# B&R Automation Studio project Teknologia25 (part 8)

#### Main.cpp - Init, cyclic, exit code
```cpp
#include <bur/plctypes.h>
#ifdef _DEFAULT_INCLUDES
	#include <AsDefault.h>
#endif
#include <cosyWriteApi.h>
#include <cosyReadApi.h>
#include <stdint.h>
#include <stdio.h>
#include <parson.h>
#include <moApi.h>

#define TRUE 1
#define FALSE 0
#define booltoa(x) ((x)?"true":"false")

void cosyExample_ReadConfig(UDINT);
void cosyExample_WriteConfig(UDINT);
int json_get_array_memberStr(UDINT,UDINT,UDINT,int,UDINT);
int json_get_array_memberNumber(UDINT,UDINT,UDINT,int,UDINT);
int json_get_array_memberBool(UDINT,UDINT,UDINT,int,UDINT);
int json_dotget_number(UDINT,UDINT,UDINT);
unsigned long bur_heap_size = 0xffff;

void _INIT ProgramInit(void)
{
	webservice.enable = TRUE;
	webservice.pRequestHeader = (UDINT)&requestHeader;
	webservice.pRequestData = (UDINT)&request;
	webservice.requestDataSize = sizeof(request);
	webservice.pServiceName 	= (UDINT)&"conf6d.cgi"; //
	webservice.option 		= httpOPTION_HTTP_11 + httpOPTION_SERVICE_TYPE_NAME;

	webservice.pUri = (UDINT)&uri;
	webservice.uriSize = sizeof(uri);
	cosyExample_ReadConfig((UDINT)&layout);
}

void _CYCLIC ProgramCyclic(void)
{
	if(webservice.send)
	{
		webservice.send = FALSE;
	}
	else if(webservice.status == ERR_OK && webservice.phase == httpPHASE_RECEIVED && !webservice.send)
	{
		httpGetParamUrl_0.pSrc = (UDINT)&uri;
		httpGetParamUrl_0.enable = TRUE;
		httpGetParamUrl_0.pParam = (UDINT)&"cmd";
		httpGetParamUrl_0.pValue = (UDINT)&cmd;
		httpGetParamUrl_0.valueSize = sizeof(cmd);
		httpGetParamUrl(&httpGetParamUrl_0);

		if(httpGetParamUrl_0.status == ERR_OK)
		{
			httpGetParamUrl_0.enable = FALSE;
			httpGetParamUrl(&httpGetParamUrl_0);
		}

		if(brsstrcmp((UDINT)&cmd,(UDINT)&"read") == 0)
		{
			brsstrcpy((UDINT)&responseHeader.contentType,(UDINT)&"application/json");
			brsstrcpy((UDINT)&response,(UDINT)&"{\"status\":\"ok\",\"layout\":{\"x\":");
			sprintf(response,"%s%i,\"y\":%i,\"segments\":[",response,layout.Xcount,layout.Ycount);
			for(int i = 0; i < layout.SegmentCount; ++i)
			{
				sprintf(response,"%s{\"x\":%i,\"y\":%i,\"name\":\"%s\",\"IsMaster\":%s}",response,layout.Segments[i].x,layout.Segments[i].y,layout.Segments[i].Name,booltoa(layout.Segments[i].IsMaster));
				if(i != (layout.SegmentCount-1))
				{
					brsstrcat((UDINT)&response,(UDINT)&",");
				}
			}
			brsstrcat((UDINT)&response,(UDINT)&"]}}");
		}
		else if(brsstrcmp((UDINT)&cmd,(UDINT)&"write") == 0)
		{
			brsstrcpy((UDINT)&responseHeader.contentType,(UDINT)&"application/json");
			brsmemset((UDINT)&layout,0,sizeof(layout));
			json_dotget_number((UDINT)&request,(UDINT)&"x",(UDINT)&tmpREAL);
			layout.Xcount = (USINT)tmpREAL;
			json_dotget_number((UDINT)&request,(UDINT)&"y",(UDINT)&tmpREAL);
			layout.Ycount = (USINT)tmpREAL;
			layout.SegmentCount = 0;
			for(int i = 0; i < 255; ++i)
			{
				if(json_get_array_memberNumber((UDINT)&request,(UDINT)&"segments",(UDINT)&"x",i,(UDINT)&tmpREAL) >= 0)
				{
					layout.Segments[i].x = (INT)tmpREAL;
					json_get_array_memberNumber((UDINT)&request,(UDINT)&"segments",(UDINT)&"y",i,(UDINT)&tmpREAL);
					layout.Segments[i].y = (INT)tmpREAL;
					json_get_array_memberBool((UDINT)&request,(UDINT)&"segments",(UDINT)&"IsMaster",i,(UDINT)&layout.Segments[i].IsMaster);
					layout.SegmentCount++;
				}
				else
				{
					break;
				}
			}
			cosyExample_WriteConfig((UDINT)&layout);
			brsstrcpy((UDINT)&response,(UDINT)&"{\"status\":\"ok\"}");
		}
		else
		{
			brsstrcpy((UDINT)&responseHeader.contentType,(UDINT)&"image/svg+xml"); //
			httpDecodeBase64_0.enable = TRUE;
			httpDecodeBase64_0.destSize = sizeof(response);
			httpDecodeBase64_0.pDest = (UDINT)&response;
			httpDecodeBase64_0.pSrc = (UDINT)&svgResource;
			httpDecodeBase64_0.srcLen = brsstrlen((UDINT)&svgResource);
			httpDecodeBase64(&httpDecodeBase64_0);
		}
		brsstrcpy((UDINT)&responseHeader.userLine[0].name,(UDINT)&"Cross-Origin-Resource-Policy");
		brsstrcpy((UDINT)&responseHeader.userLine[0].value,(UDINT)&"cross-origin");
		brsstrcpy((UDINT)&responseHeader.userLine[1].name,(UDINT)&"Access-Control-Allow-Origin");
		brsstrcpy((UDINT)&responseHeader.userLine[1].value,(UDINT)&"*");
		webservice.pResponseHeader = (UDINT)&responseHeader;
		webservice.pResponseData = (UDINT)&response;
		webservice.responseDataLen 	= brsstrlen((UDINT)&response);
		webservice.send = TRUE;
	}
	httpService(&webservice);

}

/* In the example code, error handling was deliberately omitted. */
void cosyExample_ReadConfig(UDINT context)
{
	Layout_typ myLayout;
	brsmemcpy((UDINT)&myLayout,context,sizeof(myLayout));
	uint32_t intValue = 0;
	BOOL boolValue = FALSE;
	char strValue[130];
	char tempID[60];
	COSY_H hCosy = cosyOpenElement("System/mapp6D/LayoutConfiguration", "Layout6D_1");
	cosyGetPropertyValue(hCosy, "Segments/SegRow", "USINT", sizeof(intValue),&intValue, NULL);
	myLayout.Ycount = (USINT)intValue;
	cosyGetPropertyValue(hCosy, "Segments/SegCol", "USINT", sizeof(intValue),&intValue, NULL);
	myLayout.Xcount = (USINT)intValue;
	myLayout.SegmentCount = 0;
	for(int i = 0; i < 255; ++i)
	{
		sprintf(tempID,"Segments/Segment[%i]/X",(i+1));
		if(cosyGetPropertyValue(hCosy,tempID, "INT", sizeof(intValue),&intValue, NULL))
		{
			myLayout.Segments[i].x = (INT)intValue;
			sprintf(tempID,"Segments/Segment[%i]/Y",(i+1));
			cosyGetPropertyValue(hCosy,tempID, "INT", sizeof(intValue),&intValue, NULL);
			myLayout.Segments[i].y = (INT)intValue;
			sprintf(tempID,"Segments/Segment[%i]/Name",(i+1));
			cosyGetPropertyValue(hCosy,tempID, "STRING", sizeof(strValue),&strValue, NULL);
			brsstrcpy((UDINT)&myLayout.Segments[i].Name,(UDINT)&strValue);
			sprintf(tempID,"Segments/Segment[%i]/IsMaster",(i+1));
			cosyGetPropertyValue(hCosy,tempID, "BOOL", sizeof(intValue),&intValue, NULL);
			myLayout.Segments[i].IsMaster = (BOOL)intValue;
			myLayout.SegmentCount++;
		}
		else
		{
			break;
		}
	}
	cosyCloseElement(hCosy);
	brsmemcpy(context,(UDINT)&myLayout,sizeof(myLayout));
}
void cosyExample_WriteConfig(UDINT context)
{
	Layout_typ myLayout;
	uint32_t intValue = 0;
	BOOL boolValue = FALSE;
	USINT usintValue = 0;
	USINT i = 0;
	INT tempINT = 0;
	DINT tempDINT = 0;
	char segmentName[60];
	brsmemcpy((UDINT)&myLayout,context,sizeof(myLayout));
	COSY_H hCosy = cosyOpenElement("System/mapp6D/LayoutConfiguration", "Layout6D_1");
	if(hCosy != NULL)
	{
		cosySetProperty(hCosy, "Segments/SegCol", "USINT", &myLayout.Xcount, sizeof(myLayout.Xcount));
		cosySetProperty(hCosy, "Segments/SegRow", "USINT", &myLayout.Ycount, sizeof(myLayout.Ycount));
		for(i = 0; i < 255; ++i)
		{
			sprintf(segmentName,"Segments/Segment[%i]",(i+1));
			if(!cosyDeleteMember(hCosy,segmentName,COSY_TIMEOUT_NO_WAIT))
			{
				break;
			}
		}
		for(i = 0; i < myLayout.SegmentCount; ++i)
		{
			sprintf(segmentName,"Segments/Segment[%i]",(i+1));
			cosyAddGroup(hCosy, segmentName, NULL);

			sprintf(segmentName,"Segments/Segment[%i]/Y",(i+1));
			cosySetProperty(hCosy, segmentName, "INT", &myLayout.Segments[i].y, sizeof(myLayout.Segments[i].y));
			sprintf(segmentName,"Segments/Segment[%i]/X",(i+1));
			cosySetProperty(hCosy, segmentName, "INT", &myLayout.Segments[i].x, sizeof(myLayout.Segments[i].x));
			sprintf(segmentName,"Segments/Segment[%i]/Name",(i+1));
			cosySetProperty(hCosy, segmentName, "STRING", &myLayout.Segments[i].Name, sizeof(myLayout.Segments[i].Name));
			sprintf(segmentName,"Segments/Segment[%i]/IsMaster",(i+1));

			cosySetProperty(hCosy, segmentName, "BOOL", &myLayout.Segments[i].IsMaster, 0);

			sprintf(segmentName,"Segments/Segment[%i]/PowerSectorName",(i+1));
			cosySetProperty(hCosy, segmentName, "STRING", "", 0);
			sprintf(segmentName,"Segments/Segment[%i]/Gaps",(i+1));
			cosyAddGroup(hCosy, segmentName, NULL);
			tempDINT = 0;
			sprintf(segmentName,"Segments/Segment[%i]/Gaps/Left",(i+1));
			cosySetProperty(hCosy, segmentName, "DINT", &tempDINT,sizeof(tempDINT));
			sprintf(segmentName,"Segments/Segment[%i]/Gaps/Bottom",(i+1));
			cosySetProperty(hCosy, segmentName, "DINT", &tempDINT,sizeof(tempDINT));
			sprintf(segmentName,"Segments/Segment[%i]/Gaps/Right",(i+1));
			cosySetProperty(hCosy, segmentName, "DINT", &tempDINT,sizeof(tempDINT));
			sprintf(segmentName,"Segments/Segment[%i]/Gaps/Top",(i+1));
			cosySetProperty(hCosy, segmentName, "DINT", &tempDINT,sizeof(tempDINT));
		}
		cosySaveElement(hCosy);
		cosyCloseElement(hCosy);
	}
}

int json_get_array_memberStr(UDINT data,UDINT arraystr,UDINT target,int index,UDINT result)
{
	/*TODO: Add your code here*/
	char buf[8000];
	char member[32];
	char memberValue[256];
	brsstrcpy((UDINT)&buf,data);

	JSON_Value *jsonRoot = json_parse_string(buf);
	brsstrcpy((UDINT)&member,arraystr);
	int retVal = 0;
	if(jsonRoot != NULL)
	{
		JSON_Array *arr = json_object_dotget_array(json_object(jsonRoot), member);
		if(arr != NULL)
		{
			JSON_Object *arrValue = json_array_get_object(arr,(size_t)index);
			if(arrValue != NULL)
			{
				const char *tempStr = NULL;
				char test[30];
				brsstrcpy((UDINT)&test,target);
				tempStr = json_object_dotget_string(arrValue,test);
				if(tempStr != NULL)
				{
					brsstrcpy(result,(UDINT)tempStr);
					retVal = 0;
				}
				else
				{
					retVal = -1;
				}
			}
			else
			{
				retVal = -1;
			}
		}
		else
		{
			retVal = -1;
		}
	}
	else
	{
		retVal = -1;
	}

	json_value_free(jsonRoot);
	return retVal;
}

int json_get_array_memberNumber(UDINT data,UDINT arraystr,UDINT target,int index,UDINT result)
{
	/*TODO: Add your code here*/
	char buf[8000];
	char member[32];
	char memberValue[256];
	brsstrcpy((UDINT)&buf,data);

	JSON_Value *jsonRoot = json_parse_string(buf);
	brsstrcpy((UDINT)&member,arraystr);
	int retVal = 0;
	if(jsonRoot != NULL)
	{
		JSON_Array *arr = json_object_dotget_array(json_object(jsonRoot), member);
		if(arr != NULL)
		{
			JSON_Object *arrValue = json_array_get_object(arr,(size_t)index);
			if(arrValue != NULL)
			{
				char test[30];
				brsstrcpy((UDINT)&test,target);
				double number = json_object_dotget_number(arrValue,test);
				REAL tempREAL = (REAL)number;
				brsmemcpy(result,(UDINT)&tempREAL,sizeof(tempREAL));
				//brsstrcpy(result,(UDINT)tempStr);
				retVal = 0;
			}
			else
			{
				retVal = -1;
			}
		}
		else
		{
			retVal = -1;
		}
	}
	else
	{
		retVal = -1;
	}

	json_value_free(jsonRoot);
	return retVal;
}

int json_get_array_memberBool(UDINT data,UDINT arraystr,UDINT target,int index,UDINT result)
{
	/*TODO: Add your code here*/
	char buf[8000];
	char member[32];
	char memberValue[256];
	brsstrcpy((UDINT)&buf,data);

	JSON_Value *jsonRoot = json_parse_string(buf);
	brsstrcpy((UDINT)&member,arraystr);
	int retVal = 0;
	if(jsonRoot != NULL)
	{
		JSON_Array *arr = json_object_dotget_array(json_object(jsonRoot), member);
		if(arr != NULL)
		{
			JSON_Object *arrValue = json_array_get_object(arr,(size_t)index);
			if(arrValue != NULL)
			{
				char test[30];
				brsstrcpy((UDINT)&test,target);
				int number = json_object_dotget_boolean(arrValue,test);
				BOOL tempBOOL = (BOOL)number;
				brsmemcpy(result,(UDINT)&tempBOOL,sizeof(tempBOOL));
				//brsstrcpy(result,(UDINT)tempStr);
				retVal = 0;
			}
			else
			{
				retVal = -1;
			}
		}
		else
		{
			retVal = -1;
		}
	}
	else
	{
		retVal = -1;
	}
	json_value_free(jsonRoot);
	return retVal;
}

int json_dotget_number(UDINT data,UDINT memberstr,UDINT result)
{
	/*TODO: Add your code here*/
	char buf[8000];
	char member[32];
	char memberValue[256];
	brsstrcpy((UDINT)&buf,data);

	JSON_Value *jsonRoot = json_parse_string(buf);
	brsstrcpy((UDINT)&member,memberstr);
	int retVal = -1;
	if(jsonRoot != NULL)
	{
		double temp = 0;
		temp = json_object_dotget_number(json_object(jsonRoot), member);
		REAL tempREAL = (REAL)temp;
		brsmemcpy(result,(UDINT)&tempREAL,sizeof(tempREAL));
		retVal = 0;
		//memcpy(result,(UDINT)&temp,4);

	}

	json_value_free(jsonRoot);
	return retVal;
}
```

#### Types.typ - Local data types
```iecst
TYPE
	Segment_typ : 	STRUCT
		x : INT;
		y : INT;
		IsMaster : BOOL;
		Name : STRING[20];
	END_STRUCT;
	Layout_typ : 	STRUCT
		Segments : ARRAY[0..99]OF Segment_typ;
		SegmentCount : USINT;
		Xcount : USINT;
		Ycount : USINT;
	END_STRUCT;
END_TYPE
```

#### Variables.var - Local variables
```iecst
VAR
	layout : Layout_typ;
	webservice : httpService;
	httpDecodeBase64_0 : httpDecodeBase64;
	requestHeader : httpRequestHeader_t;
	responseHeader : httpResponseHeader_t;
	svgResource : STRING[13500] := 'PHN2ZyBpZD0iNmRzdmciIHhtbG5zPSJodHRwOi8vd3d3LnczLm9yZy8yMDAwL3N2ZyIgd2lkdGg9IjYwMCIgaGVpZ2h0PSI4MjAiIHhtbDpzcGFjZT0icHJlc2VydmUiIGNvbG9yLWludGVycG9sYXRpb24tZmlsdGVycz0ic1JHQiI+Cgk8c3R5bGU+c3Zne2ZpbGw6bm9uZTsgZmlsbCAtIHJ1bGU6ZXZlbm9kZDsgZm9udCAtIHNpemU6MTJweDsgb3ZlcmZsb3c6dmlzaWJsZTsgc3Ryb2tlIC0gbGluZWNhcDpzcXVhcmU7IHN0cm9rZSAtIG1pdGVybGltaXQ6Mzt9LnNlZ21lbnQucG93ZXItb2ZmIHtmaWxsOnJnYigyNTMsIDI1MywgMjUzKTt9LnNlZ21lbnQucG93ZXItb24ge2ZpbGw6cmdiKDE0NiwgMjA4LCA4MCk7fS5zZWdtZW50LmVycm9yIHtmaWxsOnJnYigyNTIsIDIyLCAxNik7fS5zZWdtZW50ICZndDsgcmVjdCB7c3Ryb2tlOiM1OTU5NTk7c3Ryb2tlLWxpbmVjYXA6cm91bmQ7c3Ryb2tlLWxpbmVqb2luOnJvdW5kO3N0cm9rZS13aWR0aDozLjc1MDAwMDt9IC5zaHV0dGxlICZndDsgZyAmZ3Q7IHJlY3Qge3N0cm9rZTpibGFjaztzdHJva2UtbGluZWNhcDpyb3VuZDtzdHJva2UtbGluZWpvaW46cm91bmQ7c3Ryb2tlLXdpZHRoOjUuMDAwMDtmaWxsOmxpZ2h0Z3JheTt9IC5zaHV0dGxlLndhcm5pbmcgJmd0OyBnICZndDsgcmVjdCB7ZmlsbDp5ZWxsb3c7fSAuc2h1dHRsZS5lcnJvciAmZ3Q7IGcgJmd0OyByZWN0IHtmaWxsOnJlZDt9IC5zaHV0dGxlLmRpc2FibGVkICZndDsgZyAmZ3Q7IHJlY3Qge2ZpbGw6Z3JheTt9IC5zaHV0dGxlLmRpc2NvdmVyaW5nICZndDsgZyAmZ3Q7IHJlY3Qge2ZpbGw6ZGFya29yYW5nZTt9ICAuc21hbGwge2ZvbnQ6IDE1cHggc2Fucy1zZXJpZjtjb2xvcjpibGFjaztzdHJva2U6YmxhY2s7ZmlsbDpibGFjazstd2Via2l0LXVzZXItc2VsZWN0OiBub25lOyAtbXMtdXNlci1zZWxlY3Q6IG5vbmU7IHVzZXItc2VsZWN0OiBub25lO30gLnNodXR0bGV7IGN1cnNvcjpwb2ludGVyfSAuc2h1dHRsZTphY3RpdmUgJmd0OyBnICZndDsgcmVjdCB7ZmlsbDpsaWdodGJsdWU7fSAuc2h1dHRsZS50ZW1wICZndDsgZyAmZ3Q7IHJlY3Qge2ZpbGw6cmdiYSgxMjcsMTI3LDEyNywwLjEpO3N0cm9rZTpyZ2JhKDAsMCwwLDAuMSk7c3Ryb2tlLWRhc2hhcnJheToyMDt9IC5zaHV0dGxlLnRlbXAuYWN0aXZlICZndDsgZyAmZ3Q7IHJlY3Qge2ZpbGw6cmdiYSgxMjcsMCwwLDAuMSk7fTwvc3R5bGU+Cgk8cmVjdCB4PSI0OCIgeT0iMjMiIHN0eWxlPSJzdHJva2U6bGlnaHRncmF5O3N0cm9rZS13aWR0aDoxcHgiIHdpZHRoPSI0ODQiIGhlaWdodD0iMTA1Ii8+Cgk8Zm9yZWlnbk9iamVjdCB4PSIxMDAiIHk9IjM1IiAKCQkJCXdpZHRoPSI1MDAiIGhlaWdodD0iMTYwIiA+IAoJCTxkaXYgeG1sbnM9Imh0dHA6Ly93d3cudzMub3JnLzE5OTkveGh0bWwiPiAKCQkJPGxhYmVsIGZvcj0ieFNpemUiPlggRGlyZWN0aW9uPC9sYWJlbD48YnIvPgoJCQk8aW5wdXQgdHlwZT0ibnVtYmVyIiBpZD0ieFNpemUiIG5hbWU9InhTaXplIiBtaW49IjEiIG1heD0iMzAiIHZhbHVlPSIxIiAvPgkJCQoJCTwvZGl2PiAKCTwvZm9yZWlnbk9iamVjdD4gCgk8Zm9yZWlnbk9iamVjdCB4PSIyNTAiIHk9IjM1IiAKCQkJCXdpZHRoPSI1MDAiIGhlaWdodD0iMTYwIiA+IAoJCTxkaXYgeG1sbnM9Imh0dHA6Ly93d3cudzMub3JnLzE5OTkveGh0bWwiPiAKCQkJPGxhYmVsIGZvcj0ieVNpemUiPlkgRGlyZWN0aW9uPC9sYWJlbD48YnIvPgoJCQk8aW5wdXQgdHlwZT0ibnVtYmVyIiBpZD0ieVNpemUiIG5hbWU9InlTaXplIiBtaW49IjEiIG1heD0iMzAiIHZhbHVlPSIxIi8+CgkJPC9kaXY+IAoJPC9mb3JlaWduT2JqZWN0PiAKCTxmb3JlaWduT2JqZWN0IHg9IjM3NSIgeT0iMzUiIAoJCQkJd2lkdGg9IjExMCIgaGVpZ2h0PSIxNjAiID4gCgkJPGRpdiB4bWxucz0iaHR0cDovL3d3dy53My5vcmcvMTk5OS94aHRtbCI+IAoJCQk8bGFiZWwgPkFjdGl2ZSBTZWdtZW50czwvbGFiZWw+PGJyLz4KCQkJPGNlbnRlcj48bGFiZWwgaWQ9InNlZ21lbnRDb3VudCI+MDwvbGFiZWw+PC9jZW50ZXI+CgkJPC9kaXY+IAoJPC9mb3JlaWduT2JqZWN0PiAKCTxmb3JlaWduT2JqZWN0IHg9IjM2NSIgeT0iOTUiIAoJCQkJd2lkdGg9IjI1MCIgaGVpZ2h0PSIxNjAiID4gCgkJPGRpdiB4bWxucz0iaHR0cDovL3d3dy53My5vcmcvMTk5OS94aHRtbCI+IAoJCQk8YnV0dG9uIHR5cGU9ImJ1dHRvbiIgb25jbGljaz0icmVhZFBMQygpIj5SZWFkIFBMQzwvYnV0dG9uPgoJCQk8YnV0dG9uIHR5cGU9ImJ1dHRvbiIgb25jbGljaz0id3JpdGVQTEMoKSI+V3JpdGUgUExDPC9idXR0b24+CgkJPC9kaXY+IAoJPC9mb3JlaWduT2JqZWN0PiAKCTxnIGlkPSJnQXNzZW1ibHk2RF8xIiBjbGFzcz0iYXNzZW1ibHkiIHRyYW5zZm9ybT0idHJhbnNsYXRlKDUwLjAwMDAwMCA2MjAuMDAwMDAwKSI+CgkJPGcgaWQ9IkxheW91dDZEXzEiIGNsYXNzPSJsYXlvdXQiPgoJCQk8ZyBpZD0ic2VnbWVudHMiPjwvZz4KCQk8L2c+Cgk8L2c+Cgk8ZyBpZD0iY29udGV4dE1lbnUiPjwvZz4KCTxzY3JpcHQ+Ly88IVtDREFUQVsKCQl2YXIgeENvdW50ID0gZG9jdW1lbnQuZ2V0RWxlbWVudEJ5SWQoJ3hTaXplJyk7CgkJdmFyIHlDb3VudCA9IGRvY3VtZW50LmdldEVsZW1lbnRCeUlkKCd5U2l6ZScpOwoJCXZhciBzZWdtZW50cyA9IGRvY3VtZW50LmdldEVsZW1lbnRCeUlkKCdzZWdtZW50cycpOwoJCXZhciBzZWdtZW50Q291bnQgPSBkb2N1bWVudC5nZXRFbGVtZW50QnlJZCgnc2VnbWVudENvdW50Jyk7CgkJdmFyIGNvbnRleHRNZW51ID0gZG9jdW1lbnQuZ2V0RWxlbWVudEJ5SWQoJ2NvbnRleHRNZW51Jyk7CgkJdmFyIHNlZ21lbnRTaXplID0gMDsKCQl4Q291bnQuYWRkRXZlbnRMaXN0ZW5lcigiY2hhbmdlIiwgKGV2ZW50KSA9PiB7c2V0TGF5b3V0KHhDb3VudC52YWx1ZSx5Q291bnQudmFsdWUpO30pOwoJCXlDb3VudC5hZGRFdmVudExpc3RlbmVyKCJjaGFuZ2UiLCAoZXZlbnQpID0+IHtzZXRMYXlvdXQoeENvdW50LnZhbHVlLHlDb3VudC52YWx1ZSk7fSk7CgkJCgkJdmFyIGFjdGl2ZVNlZ21lbnRzID0gW107CgkJdmFyIHN2Z0VsZW0gPSBkb2N1bWVudC5nZXRFbGVtZW50QnlJZCgnNmRzdmcnKTsKCQkJCXN2Z0VsZW0uYWRkRXZlbnRMaXN0ZW5lcigibG9hZCIsICgpID0+IHsKCQkJcmVhZFBMQygpOwoJCX0pOwoJCWZ1bmN0aW9uIHJlYWRQTEMoKQoJCXsKCQkJdmFyIHhodHRwID0gbmV3IFhNTEh0dHBSZXF1ZXN0KCk7CgkJCQl4aHR0cC5vbnJlYWR5c3RhdGVjaGFuZ2UgPSBmdW5jdGlvbigpIHsKCQkJCQlpZiAodGhpcy5yZWFkeVN0YXRlID09IDQgJiYgdGhpcy5zdGF0dXMgPT0gMjAwKSB7CgkJCQkJICAgLy8gVHlwaWNhbCBhY3Rpb24gdG8gYmUgcGVyZm9ybWVkIHdoZW4gdGhlIGRvY3VtZW50IGlzIHJlYWR5OgoJCQkJCSAgIHZhciBkYXRhID0gSlNPTi5wYXJzZSh4aHR0cC5yZXNwb25zZVRleHQpOwoJCQkJCSAgIGFjdGl2ZVNlZ21lbnRzID0gW107CgkJCQkJICAgZm9yKHZhciBpID0gMDsgaSA8IGRhdGEubGF5b3V0LnNlZ21lbnRzLmxlbmd0aDsgKytpKQoJCQkJCSAgIHsKCQkJCQkJCWFjdGl2ZVNlZ21lbnRzLnB1c2goe3g6ZGF0YS5sYXlvdXQuc2VnbWVudHNbaV0ueCx5OmRhdGEubGF5b3V0LnNlZ21lbnRzW2ldLnksSXNNYXN0ZXI6ZGF0YS5sYXlvdXQuc2VnbWVudHNbaV0uSXNNYXN0ZXJ9KTsKCQkJCQkJCWlmKGRhdGEubGF5b3V0LnNlZ21lbnRzW2ldLklzTWFzdGVyKQoJCQkJCQkJewoJCQkJCQkJCXNldE1hc3RlckJ5U2VnbWVudChhY3RpdmVTZWdtZW50c1thY3RpdmVTZWdtZW50cy5sZW5ndGgtMV0pOwoJCQkJCQkJfQoJCQkJCSAgIH0KCQkJCQkgICB4Q291bnQudmFsdWUgPSBkYXRhLmxheW91dC54OwoJCQkJCSAgIHlDb3VudC52YWx1ZSA9IGRhdGEubGF5b3V0Lnk7CgkJCQkJICAgc2V0TGF5b3V0KGRhdGEubGF5b3V0LngsZGF0YS5sYXlvdXQueSk7CgkJCQkJfQoJCQkJfTsKCQkJCXhodHRwLm9wZW4oIkdFVCIsICIvY29uZjZkLmNnaT9jbWQ9cmVhZCIsIHRydWUpOwoJCQkJeGh0dHAuc2VuZCgpOwoJCX0KCQlmdW5jdGlvbiB3cml0ZVBMQygpCgkJewoJCQl2YXIgeGh0dHAgPSBuZXcgWE1MSHR0cFJlcXVlc3QoKTsKCQkJCXhodHRwLm9ucmVhZHlzdGF0ZWNoYW5nZSA9IGZ1bmN0aW9uKCkgewoJCQkJCWlmICh0aGlzLnJlYWR5U3RhdGUgPT0gNCAmJiB0aGlzLnN0YXR1cyA9PSAyMDApIHsKCQkJCQkgICAvLyBUeXBpY2FsIGFjdGlvbiB0byBiZSBwZXJmb3JtZWQgd2hlbiB0aGUgZG9jdW1lbnQgaXMgcmVhZHk6CgkJCQkJICAgdmFyIGRhdGEgPSBKU09OLnBhcnNlKHhodHRwLnJlc3BvbnNlVGV4dCk7CgkJCQkJICAgY29uc29sZS5sb2coZGF0YSk7CgkJCQkJfQoJCQkJfTsKCQkJCXhodHRwLm9wZW4oIlBPU1QiLCAiL2NvbmY2ZC5jZ2k/Y21kPXdyaXRlIiwgdHJ1ZSk7CgkJCQlhY3RpdmVTZWdtZW50cy5zb3J0KGNvbXBhcmVGbik7CgkJCQl2YXIgbWFzdGVyRWxlbWVudCA9IGRvY3VtZW50LmdldEVsZW1lbnRCeUlkKCdtYXN0ZXItdGV4dCcpOwoJCQkJaWYoIW1hc3RlckVsZW1lbnQpCgkJCQl7CgkJCQkJYWN0aXZlU2VnbWVudHNbMF0uSXNNYXN0ZXIgPSB0cnVlOwoJCQkJfQoJCQkJeGh0dHAuc2VuZChKU09OLnN0cmluZ2lmeSh7eDpwYXJzZUludCh4Q291bnQudmFsdWUpLHk6cGFyc2VJbnQoeUNvdW50LnZhbHVlKSxzZWdtZW50czphY3RpdmVTZWdtZW50c30pKTsKCQl9CgkJCgkJZnVuY3Rpb24gY29tcGFyZUZuKGEsIGIpIHsKCQkgIGlmIChhLnggPCBiLngpIHsKCQkJcmV0dXJuIC0xOwoJCSAgfWVsc2UgaWYgKGEueCA+IGIueCkgewoJCQlyZXR1cm4gMTsKCQkgIH1lbHNlIGlmIChhLnkgPCBiLnkpIHsKCQkJcmV0dXJuIC0xOwoJCSAgfWVsc2UgaWYgKGEueSA+IGIueSkgewoJCQlyZXR1cm4gMTsKCQkgIH0KCQkgIC8vIGEgbXVzdCBiZSBlcXVhbCB0byBiCgkJICByZXR1cm4gMDsKCQl9OwoJCQoJCWZ1bmN0aW9uIGNoYW5nZVN0eWxlKHRoYXQpCgkJewoJCQlpZihjb250ZXh0TWVudS5pbm5lckhUTUwgPT0gJycpCgkJCXsKCQkJCWlmKHRoYXQuY2xhc3NMaXN0WzFdID09ICdwb3dlci1vZmYnKQoJCQkJewoJCQkJCXRoYXQuY2xhc3NMaXN0LnJlbW92ZSgicG93ZXItb2ZmIik7CgkJCQkJdGhhdC5jbGFzc0xpc3QuYWRkKCJwb3dlci1vbiIpOwoJCQkJCWFjdGl2ZVNlZ21lbnRzLnB1c2goe3g6cGFyc2VJbnQodGhhdC5nZXRBdHRyaWJ1dGUoJ3Bvc2l0aW9uLXgnKSkseTpwYXJzZUludCh0aGF0LmdldEF0dHJpYnV0ZSgncG9zaXRpb24teScpKSxJc01hc3RlcjpmYWxzZX0pOwoJCQkJfQoJCQkJZWxzZQoJCQkJewoJCQkJCXRoYXQuY2xhc3NMaXN0LmFkZCgicG93ZXItb2ZmIik7CgkJCQkJdGhhdC5jbGFzc0xpc3QucmVtb3ZlKCJwb3dlci1vbiIpOwoJCQkJCXZhciByZW1vdmVJdGVtID0ge3g6dGhhdC5nZXRBdHRyaWJ1dGUoJ3Bvc2l0aW9uLXgnKSx5OnRoYXQuZ2V0QXR0cmlidXRlKCdwb3NpdGlvbi15Jyl9CgkJCQkJZm9yKHZhciBpID0gMDsgaSA8IGFjdGl2ZVNlZ21lbnRzLmxlbmd0aDsgKytpKQoJCQkJCXsKCQkJCQkJaWYoKGFjdGl2ZVNlZ21lbnRzW2ldLnggPT0gcmVtb3ZlSXRlbS54KSAmJiAoYWN0aXZlU2VnbWVudHNbaV0ueSA9PSByZW1vdmVJdGVtLnkpKQoJCQkJCQl7CgkJCQkJCQlhY3RpdmVTZWdtZW50cy5zcGxpY2UoaSwgMSk7CgkJCQkJCQlicmVhazsKCQkJCQkJfQoJCQkJCX0KCQkJCX0KCQkJfQoJCQljb250ZXh0TWVudS5pbm5lckhUTUwgPSAnJzsKCQkJc2VnbWVudENvdW50LmlubmVySFRNTCA9IGFjdGl2ZVNlZ21lbnRzLmxlbmd0aDsKCQkJCgkJfQoJCWZ1bmN0aW9uIHNldE1hc3Rlcih0aGF0KQoJCXsKCQkJdmFyIGlkeCA9IHBhcnNlSW50KHRoYXQuZ2V0QXR0cmlidXRlKCdzZWdtZW50LWluZGV4JykpOwoJCQl2YXIgdGFyZ2V0SWQgPSB0aGF0LmdldEF0dHJpYnV0ZSgndGFyZ2V0LWlkJyk7CgkJCWZvcih2YXIgaSA9IDA7IGkgPCBhY3RpdmVTZWdtZW50cy5sZW5ndGg7ICsraSkKCQkJewoJCQkJYWN0aXZlU2VnbWVudHNbaV1bIklzTWFzdGVyIl0gPSBmYWxzZTsKCQkJfQoJCQlhY3RpdmVTZWdtZW50c1tpZHhdWyJJc01hc3RlciJdID0gdHJ1ZTsKCQkJY29udGV4dE1lbnUuaW5uZXJIVE1MID0gJyc7CgkJCQoJCQl2YXIgdGFyZ2V0ID0gZG9jdW1lbnQuZ2V0RWxlbWVudEJ5SWQodGFyZ2V0SWQpOwoJCQl2YXIgbWFzdGVyVGV4dCA9IGRvY3VtZW50LmdldEVsZW1lbnRCeUlkKCdtYXN0ZXItdGV4dCcpOwoJCQlpZihtYXN0ZXJUZXh0KQoJCQl7CgkJCQltYXN0ZXJUZXh0LnBhcmVudEVsZW1lbnQucmVtb3ZlQ2hpbGQobWFzdGVyVGV4dCk7CgkJCX0KCQkJdmFyIHRleHQgPSBkb2N1bWVudC5jcmVhdGVFbGVtZW50TlMoImh0dHA6Ly93d3cudzMub3JnLzIwMDAvc3ZnIiwgInRleHQiKTsKCQkJdGV4dC5zZXRBdHRyaWJ1dGUoJ3gnLDUpOwoJCQl0ZXh0LnNldEF0dHJpYnV0ZSgneScsMTgpOwoJCQl0ZXh0LnNldEF0dHJpYnV0ZSgnc3R5bGUnLCdmaWxsOndoaXRlO2ZvbnQtc2l6ZToxOHB4OycpOwoJCQl0ZXh0LnNldEF0dHJpYnV0ZSgnaWQnLCdtYXN0ZXItdGV4dCcpOwoJCQl0ZXh0LmlubmVySFRNTCA9ICdNJzsKCQkJdGFyZ2V0LmFwcGVuZENoaWxkKHRleHQpOwoJCX0KCQkKCQlmdW5jdGlvbiBzZXRNYXN0ZXJCeVNlZ21lbnQoc2VnbWVudCkKCQl7CgkJCXZhciBzZWxlY3RlZFNlZ21lbnRzID0gZG9jdW1lbnQuZ2V0RWxlbWVudHNCeUNsYXNzTmFtZSgnc2VnbWVudCBwb3dlci1vbicpOwoJCQlmb3IodmFyIGkgPSAwOyBpIDwgc2VsZWN0ZWRTZWdtZW50cy5sZW5ndGg7ICsraSkKCQkJewoJCQkJaWYoKHBhcnNlSW50KHNlbGVjdGVkU2VnbWVudHNbaV0uZ2V0QXR0cmlidXRlKCdwb3NpdGlvbi14JykpID09IHNlZ21lbnQueCkgJiYgKHBhcnNlSW50KHNlbGVjdGVkU2VnbWVudHNbaV0uZ2V0QXR0cmlidXRlKCdwb3NpdGlvbi15JykpID09IHNlZ21lbnQueSkpCgkJCQl7CgkJCQkJdmFyIG1hc3RlclRleHQgPSBkb2N1bWVudC5nZXRFbGVtZW50QnlJZCgnbWFzdGVyLXRleHQnKTsKCQkJCQlpZihtYXN0ZXJUZXh0KQoJCQkJCXsKCQkJCQkJbWFzdGVyVGV4dC5wYXJlbnRFbGVtZW50LnJlbW92ZUNoaWxkKG1hc3RlclRleHQpOwoJCQkJCX0KCQkJCQl2YXIgdGV4dCA9IGRvY3VtZW50LmNyZWF0ZUVsZW1lbnROUygiaHR0cDovL3d3dy53My5vcmcvMjAwMC9zdmciLCAidGV4dCIpOwoJCQkJCXRleHQuc2V0QXR0cmlidXRlKCd4Jyw1KTsKCQkJCQl0ZXh0LnNldEF0dHJpYnV0ZSgneScsMTgpOwoJCQkJCXRleHQuc2V0QXR0cmlidXRlKCdzdHlsZScsJ2ZpbGw6d2hpdGU7Zm9udC1zaXplOjE4cHg7Jyk7CgkJCQkJdGV4dC5zZXRBdHRyaWJ1dGUoJ2lkJywnbWFzdGVyLXRleHQnKTsKCQkJCQl0ZXh0LmlubmVySFRNTCA9ICdNJzsKCQkJCQlzZWxlY3RlZFNlZ21lbnRzW2ldLmFwcGVuZENoaWxkKHRleHQpOwoJCQkJCWJyZWFrOwoJCQkJfQoJCQl9CgkJfQoJCQoJCWZ1bmN0aW9uIGFkZENvbnRleHRtZW51KGV2ZW50KQoJCXsKCQkJdmFyIHNlZ21lbnRBY3RpdmUgPSBmYWxzZTsKCQkJdmFyIHNlZ21lbnRJbmRleCA9IDA7CgkJCWZvcih2YXIgaSA9IDA7IGkgPCBhY3RpdmVTZWdtZW50cy5sZW5ndGg7ICsraSkKCQkJewoJCQkJaWYoZXZlbnQudGFyZ2V0LnBhcmVudEVsZW1lbnQuZ2V0QXR0cmlidXRlKCdwb3NpdGlvbi14JykgPT0gYWN0aXZlU2VnbWVudHNbaV0ueCAmJiBldmVudC50YXJnZXQucGFyZW50RWxlbWVudC5nZXRBdHRyaWJ1dGUoJ3Bvc2l0aW9uLXknKSA9PSBhY3RpdmVTZWdtZW50c1tpXS55KQoJCQkJewoJCQkJCXNlZ21lbnRBY3RpdmUgPSB0cnVlOwoJCQkJCXNlZ21lbnRJbmRleCA9IGk7CgkJCQkJc2VnbWVudElkID0gZXZlbnQudGFyZ2V0LnBhcmVudEVsZW1lbnQuZ2V0QXR0cmlidXRlKCdpZCcpOwoJCQkJCWJyZWFrOwoJCQkJfQoJCQl9CgkJCWlmKGV2ZW50LnByZXZlbnREZWZhdWx0ICE9IHVuZGVmaW5lZCkKCQkJICBldmVudC5wcmV2ZW50RGVmYXVsdCgpOwoJCQkgaWYoZXZlbnQuc3RvcFByb3BhZ2F0aW9uICE9IHVuZGVmaW5lZCkKCQkJICBldmVudC5zdG9wUHJvcGFnYXRpb24oKTsKCQkJIGlmKHNlZ21lbnRBY3RpdmUpCgkJCSB7CgkJCQl2YXIgY21ZID0gZXZlbnQueS0xMDUvMjsKCQkJCWNvbnRleHRNZW51LmlubmVySFRNTCA9IGA8cmVjdCB4PSIke2V2ZW50Lnh9IiB5PSIke2NtWX0iIHN0eWxlPSJzdHJva2U6bGlnaHRncmF5O3N0cm9rZS13aWR0aDoxcHg7ZmlsbDp3aGl0ZTsiIHdpZHRoPSIxMDAiIGhlaWdodD0iMTA1Ii8+CgkJCSA8Zm9yZWlnbk9iamVjdCB4PSIke2V2ZW50LngrMn0iIHk9IiR7Y21ZfSIgCgkJCQkJCXdpZHRoPSI5NiIgaGVpZ2h0PSIxMDEiID4gCgkJCQkJCTxkaXYgeG1sbnM9Imh0dHA6Ly93d3cudzMub3JnLzE5OTkveGh0bWwiPiAKCQkJCQkJCTxidXR0b24gdHlwZT0iYnV0dG9uIiBvbmNsaWNrPSJzZXRNYXN0ZXIodGhpcykiIHNlZ21lbnQtaW5kZXg9IiR7c2VnbWVudEluZGV4fSIgdGFyZ2V0LWlkPSIke3NlZ21lbnRJZH0iPlNldCBhcyBNYXN0ZXI8L2J1dHRvbj4KCQkJCQkJPC9kaXY+IAoJCQkgPC9mb3JlaWduT2JqZWN0PiBgOwoJCQkgfQoJCX0KCQlmdW5jdGlvbiBzZXRMYXlvdXQoeCx5KQoJCXsKCQkJc2VnbWVudHMuaW5uZXJIVE1MID0gJyc7CgkJCXNlZ21lbnRTaXplID0gNDgwL3k7CgkJCWlmKHBhcnNlSW50KHgpID4gcGFyc2VJbnQoeSkpCgkJCXsKCQkJCXNlZ21lbnRTaXplID0gNDgwL3g7CgkJCX0KCQkJdmFyIHNlZ21lbnRDb3VudGVyID0gMTsKCQkJdmFyIGR5bkhXID0gJyc7CgkJCWZvcih2YXIgaSA9IDA7IGkgPCBhY3RpdmVTZWdtZW50cy5sZW5ndGg7ICsraSkKCQkJewoJCQkJaWYoKHBhcnNlSW50KGFjdGl2ZVNlZ21lbnRzW2ldLngpKzEpID4gcGFyc2VJbnQoeCkpCgkJCQl7CgkJCQkJYWN0aXZlU2VnbWVudHMuc3BsaWNlKGksMSk7CgkJCQkJaSA9IDA7CgkJCQkJY29udGludWU7CgkJCQl9CgkJCQlpZigocGFyc2VJbnQoYWN0aXZlU2VnbWVudHNbaV0ueSkrMSkgPiBwYXJzZUludCh5KSkKCQkJCXsKCQkJCQlhY3RpdmVTZWdtZW50cy5zcGxpY2UoaSwxKTsKCQkJCQlpID0gMDsKCQkJCQljb250aW51ZTsKCQkJCX0KCQkJfQoJCQlmb3IodmFyIGkgPSAwOyBpIDwgeDsgKytpKQoJCQl7CgkJCQlmb3IodmFyIGogPSAwOyBqIDwgeTsgKytqKQoJCQkJewoJCQkJCXZhciBhY3RpdmUgPSBmYWxzZTsKCQkJCQlmb3IodmFyIGsgPSAwOyBrIDwgYWN0aXZlU2VnbWVudHMubGVuZ3RoOyArK2spCgkJCQkJewoJCQkJCQlpZihhY3RpdmVTZWdtZW50c1trXS54ID09IGkgJiYgYWN0aXZlU2VnbWVudHNba10ueSA9PSBqKQoJCQkJCQl7CgkJCQkJCQlhY3RpdmUgPSB0cnVlOwoJCQkJCQkJYnJlYWs7CgkJCQkJCX0KCQkJCQl9CgkJCQkJZHluSFcgKz0gYAoJCQkJCTxnIGlkPSJzZWdtZW50XyR7c2VnbWVudENvdW50ZXJ9IiBjbGFzcz0ic2VnbWVudCBwb3dlci0ke2FjdGl2ZSA/ICdvbicgOiAnb2ZmJ30iIHRyYW5zZm9ybT0idHJhbnNsYXRlKCR7c2VnbWVudFNpemUqaX0gLSR7c2VnbWVudFNpemUqKGorMSl9KSIgcG9zaXRpb24teD0iJHtpfSIgcG9zaXRpb24teT0iJHtqfSIgbWFzdGVyPSJ0cnVlIiBvbmNsaWNrPSJjaGFuZ2VTdHlsZSh0aGlzKSIgb25jb250ZXh0bWVudT0iYWRkQ29udGV4dG1lbnUoZXZlbnQpIj4KCQkJCQkJPHJlY3QgeD0iMS44NzUiIHk9IjEuODc1IiB3aWR0aD0iJHtzZWdtZW50U2l6ZX0iIGhlaWdodD0iJHtzZWdtZW50U2l6ZX0iIHJ4PSIzLjc1IiByeT0iMy43NSIvPgoJCQkJCTwvZz5gOwoJCQkJCXNlZ21lbnRDb3VudGVyKys7CgkJCQl9CgkJCX0KCQkJc2VnbWVudHMuaW5uZXJIVE1MID0gZHluSFc7CgkJCXNlZ21lbnRDb3VudC5pbm5lckhUTUwgPSBhY3RpdmVTZWdtZW50cy5sZW5ndGg7CgkJfQoJLy9dXT4KCTwvc2NyaXB0Pgo8L3N2Zz4=';
	response : STRING[13500];
	request : STRING[4000];
	uri : STRING[200];
	httpGetParamUrl_0 : httpGetParamUrl;
	cmd : STRING[80];
	tmpREAL : REAL;
	jkiTest : BOOL;
	state : USINT;
	tempSTR : STRING[80];
END_VAR
```

#### cosyApi.h
```c
/*
 * Configuration System (COSY) API
 *
 * The configuration system provides a generic mechanism to configure object instances of any type. An object
 * itself is described by a set of attributes. Thus an object configuration, represented by a COSY-element, is an
 * assembly of properties, with each property being represented by a key-/value pair. For contextual separation
 * of information, properties may be grouped hierarchically. To be able to save the configuration data permanently,
 * COSY offers the possibility to save elements non-volatile.
 *
 * COSY, as an administration of configuration elements, provides read-/write-access to its COSY-elements. For further
 * documentation see 'cosyWriteApi.h' and 'cosyReadApi.h'.
 *
 * Mind that COSY is operating on UTF encoded strings. So any function granting write access to COSY will fail
 * in case of wrong input parameter string encoding.
 *
 * COSY-element:
 * An element is uniquely identified by its path-name representing a full qualified name (fqn).
 * The fqn is divided into a location- and id-part separated by the '/' delimiter character. Further, the location-part
 * may be subdivided using the '/' delimiter character for hierarchy purpose. An element consists of groups, and
 * properties. Each group again may be organised in sub-groups and properties.
 *
 * Notation:
 * fqn := <location>/<id> with location := <arg1>/<arg2>/<arg3>/... and id := <arg>
 *
 * Sample:
 * fqn := "GMC/Axis1" with location := "GMC" and id := "Axis1"
 *
 * In addition, each element is reporting a certain type and technologyPackage. Both attributes are specified as
 * mandatory, classifying a COSY element for custom purpose.
 *
 * COSY-element type:
 * The type classifies an element. Mind that an element (uniquely specified by its location and id) of different types
 * is prohibited.
 *
 * Sample:
 * fqn := "GMC/Axis1" of type := "singleAxis" (ok)
 * fqn := "GMC/Axis1" of type := "multiAxis"  (failure)
 * fqn := "GMC/Axis2" of type := "multiAxis"  (ok)
 *
 * COSY-element technologyPackage:
 * A technologyPackage is closely related to a namespace, aggregating elements for custom specific pupose.
 *
 * COSY-element property:
 * A property is defined as a key-/value pair describing a certain attribute. Mind that a property can not be deleted on
 * demand, although it can be created.
 *
 * COSY-element group:
 * A group may be used for contextual separation of information. Mind that a group can not be deleted on demand,
 * although it can be created.
 *
 * Non-volatile COSY Element:
 * Non-volatile COSY elements are preserved across reboots. A COSY element can be saved non-volatile per
 * cosySaveElement() - Note: COSY elements transferred with the project are already non-volatile. If a non-volatile
 * element is closed, an implicit save is performed.
 * Since saving is done asynchronously, the save status can be read with cosyGetElementSaveStatus().
 */

#ifndef _COSY_API_H_
#define _COSY_API_H_

#include <stdbool.h>

#ifdef __cplusplus
extern "C" {
#endif

/* Handle for accessing a COSY element */
typedef struct COSY* COSY_H;

/*
 * Open an existing COSY element by its 'location' and 'id'.
 * Return the handle of the COSY element on success, else NULL on failure (e.g. non existing).
 *
 * Note:
 * A COSY element can be opened multiple times.
 */
COSY_H cosyOpenElement(const char* location, const char* id);

/*
 * Open an existing COSY element by its 'fqn'.
 * Return the handle of the COSY element on success, else NULL on failure (e.g. non existing).
 *
 * Note:
 * A COSY element can be opened multiple times.
 */
COSY_H cosyOpenElementByFqn(const char* fqn);

/*
 * Close a COSY element by its handle 'hCosy'.
 * Non-volatile Elements are automatically saved.
 * Return true on success, false on failure.
 */
bool cosyCloseElement(COSY_H hCosy);

/*
 * Save the COSY element specified by 'hCosy' non-volatile.
 * Return true on success, false on failure (e.g. diagnose mode).
 *
 * Note:
 * Saving a element is done asynchronously, therefore the current save status can be read out via
 * cosyGetElementSaveStatus(). Non-volatile elements are automatically saved on closing.
 */
bool cosySaveElement(COSY_H hCosy);

/*
 * Get the save status of a COSY element specified by 'hCosy'.
 * Returns the current save status:
 *   0 - the element is up to date.
 * > 0 - the non-volatile element has been changed since the last save, or there is currently a save job running.
 * < 0 - saving the element failed.
 * The error status (< 0) can be reset by modifying and saving again.
 */
int cosyGetElementSaveStatus(COSY_H hCosy);

/*
 * Evaluate if the COSY element specified by 'hCosy' is non-volatile.
 * Return true if non-volatile, false if not.
 */
bool cosyIsElementNonVolatile(COSY_H hCosy);

/*
 * Evaluate if the COSY element specified by 'hCosy' has been changed since the last save.
 * A element is dirty until it is saved again (cosySaveElement()).
 * Return true if element is dirty (only if the element is non-volatile), false if not.
 */
bool cosyIsElementDirty(COSY_H hCosy);

#ifdef __cplusplus
}
#endif

#endif
```

#### cosyReadApi.h
```c
/*
 * Configuration System (COSY) API
 *
 * This API provides functionality for accessing element member information. For reading purpose
 * element members, that can be properties as well as a groups, can be iterated too.
 *
 * For more information regarding the identification of a COSY element see cosyApi.h
 */

#ifndef _COSY_READ_API_H_
#define _COSY_READ_API_H_

#include <cosyApi.h>
#include <stdbool.h>
#include <stdint.h>
#include <stddef.h>

#ifdef __cplusplus
extern "C" {
#endif

/* COSY iterate flags */
enum COSY_ITERATE_FLAGS
{
	/* Iterate over element members of the given element non recursively */
	COSY_ITERATE_DEFAULT = 0,
	/* Iterate over element members of a given element recursively */
	COSY_ITERATE_SUB_MEMBER = 1
};

/*
 * Prototype for COSY iteration callback, that will be invoked for each existing element, whereof
 * 'context' is the user argument that will be hand over from cosyIterateElements and 'hCosy' is
 * the handle of the COSY element currently processed.
 * Return true to continue iteration, or false to stop iteration.
 *
 * Mind:
 * Within iteration context, elements must not be added or removed.
 */
typedef bool (*COSY_ITERATE_FP)(uintptr_t context, COSY_H hCosy);

/*
 * Prototype for COSY iteration callback, that will be invoked for each existing element member, whereof
 * 'context' is the user argument that will be hand over from cosyIterateMembers, 'hCosy' is the handle
 * of the COSY element currently processed, 'id' is the path information of the dedicated member
 * as UTF8 encoded string and 'memberType' is the member itself (group or property) as UTF8 encoded string.
 * Return true to continue iteration, or false to stop iteration.
 *
 * Mind:
 * Within iteration context, element members of the same iteration depth must not be added or removed.
 */
typedef bool (*COSY_ITERATE_MEMBERS_FP)(uintptr_t context, COSY_H hCosy, const char* id, const char* memberType);

/*
 * Get the location of the COSY element by 'hCosy'.
 * Return the address of the UTF8 encoded string on success, else NULL on failure.
 */
const char* cosyGetElementLocation(COSY_H hCosy);

/*
 * Get the id of the COSY element by 'hCosy'.
 * Return the address of the UTF8 encoded  string on success, else NULL on failure.
 */
const char* cosyGetElementId(COSY_H hCosy);

/*
 * Get the type of the COSY element by 'hCosy'.
 * Return the address of the UTF8 encoded string on success, else NULL on failure.
 */
const char* cosyGetElementType(COSY_H hCosy);

/* Get the technology package of the COSY element by 'hCosy'.
 * Return the address of the UTF8 encoded string on success, else NULL on failure.
 */
const char* cosyGetElementTechnologyPackage(COSY_H hCosy);

/*
 * Get the value of the group by 'id' of the COSY element by 'hCosy'.
 * Return the address of the UTF8 encoded string on success, else NULL on failure.
 */
const char* cosyGetGroupValue(COSY_H hCosy, const char* id);

/*
 * Get the type of the property by 'id' of the COSY element by 'hCosy'.
 * Return the address of the UTF8 encoded string on success, else NULL on failure.
 *
 * Mind:
 * The type information correlates with the 'iecType' described for cosyGetPropertyType.
 * It can be either the UTF8 encoded string of an IEC-Type (see iecType.h) or "BLOB" for any
 * raw data.
 */
const char* cosyGetPropertyType(COSY_H hCosy, const char* id);

/*
 * Get the value of the property by 'id' and 'iecType' of the COSY element by 'hCosy', whereof 'bytesToRead'
 * specify the size of 'pValue' in byte. 'pValueSize' is an output parameter being set on success to indicate the
 * minimum required size of byte for 'pValue'.
 * Return true on succeess, or false on failure.
 *
 * Mind:
 * In order to determine the proper size of byte by 'pValueSize' of the property value being requested,
 * 'pValue' can be set to NULL.
 *
 * Although the property is identified by its path information by 'id', the 'iecType' is mandatory
 * to interpret the 'pValue' according to the mapping table correctly.
 *
 * Convention:
 * According to the mapping table the 'pValue' is interpreted differently.
 *
 * pValue       |   bytesToRead         |   iecType
 * -------------|-----------------------|-----------
 * uint32_t     |   sizeof(uint32_t)    |   BOOL, SINT, INT, DINT, USINT, UINT, UDINT, BYTE, WORD, DWORD
 * char*        |   N bytes             |   REAL, LREAL, STRING, TIME, DATE, DATE_AND_TIME, TIME_OF_DAY
 * ----------------------------------------------------------------------------------------------
 * void*        |   N bytes             |   BLOB
 *
 * Unsupported IEC data types (see iecType.h):
 * ULINT, LWORD, WSTRING, OCTET, LINT
 */
bool cosyGetPropertyValue(COSY_H hCosy, const char* id, const char* iecType, size_t bytesToRead, void* pValue,
                          size_t* pValueSize);

/*
 * Get the size as output parameter 'pValueSize' of the property by 'id' of the COSY element
 * by 'hCosy'.
 * Return true on success, else false on failure.
 */
bool cosyGetPropertySize(COSY_H hCosy, const char* id, size_t* pValueSize);

/*
 * Iterate over COSY elements and invoke the user callback by 'fpIterate' with the user argument
 * 'context'. Set 'elementTypeFilter' to NULL to iterate over all elements, or set a value for
 * 'elementTypeFilter' to narrow the iteration down.
 * Return true on success, else false on failure.
 */
bool cosyIterateElements(COSY_ITERATE_FP fpIterate, uintptr_t context, const char* elementTypeFilter);

/*
 * Iterate over members of the COSY element by 'hCosy' and invoke the user callback by 'fpIterate' with
 * the user argument by 'context' for each member. Set 'startId' to NULL to start iteration from the first
 * member, else set a value for 'startId' to start iteration from a dedicated element member.
 * Further set 'flags' according to COSY_ITERATE_FLAGS to iterate recursively or not.
 * Return true on success, else false on failure.
 */
bool cosyIterateMembers(COSY_H hCosy, const char* startId, enum COSY_ITERATE_FLAGS flags,
                        COSY_ITERATE_MEMBERS_FP fpIterate, uintptr_t context);

/*
 * Gets the version of a COSY element by 'hCosy'.
 * Return the address of the UTF8 encoded string on success, else NULL on failure.
 */
const char* cosyGetElementVersion(COSY_H hCosy);

#if AR_CORE
#include <private/cosyReadApiP.h>
#endif

#ifdef __cplusplus
}
#endif

#endif
```

#### cosyWriteApi.h
```c
/*
 * Configuration System (COSY) API
 *
 * This API provides functionality for creating and destroying COSY elements and its members.
 * Element members can be properties as well as a groups, whereof each group can aggregate
 * properties again as well as sub groups.
 *
 * For more information regarding the identification of a COSY element see cosyApi.h
 */

#ifndef _COSY_WRITE_API_H_
#define _COSY_WRITE_API_H_

#include <cosyApi.h>
#include <stdbool.h>
#include <stdint.h>
#include <stddef.h>

#ifdef __cplusplus
extern "C" {
#endif

/* timeout behaviour defines */
#define COSY_TIMEOUT_NO_WAIT 0
#define COSY_TIMEOUT_WAIT_FOREVER 0xFFFFFFFF

/*
 * Create a new COSY element with a unique 'location' and 'id'. Both values are
 * aggregated to a fqn (see cosyApi.h) identifying the element. For the purpose of
 * detailed element specification, 'type' and 'technologyPackage' are mandatory to be set.
 * Return the handle of the COSY element on success, else NULL on failure.
 *
 * Example: fqn:= "System/GMC/Axis", where location:= "System/GMC" and id:= "Axis"
 */
COSY_H cosyCreateElement(const char* location, const char* id, const char* type, const char* technologyPackage);

/*
 * Destroy a COSY element by its 'location' and 'id'.
 * Return true on success, else false on failure.
 *
 * Mind:
 * An element with all its members will be destroyed synchronously. Saved non-volatile data are removed asynchronously.
 */
bool cosyDestroyElement(const char* location, const char* id);

/*
 * Add a group by 'id' and 'value' to a COSY element by 'hCosy'.
 * Return true on success, else false on failure.
 *
 * In case of 'id' is representing a path to a subgroup, like id:= "g1/g2/g3", all parent groups
 * will be created.
 */
bool cosyAddGroup(COSY_H hCosy, const char* id, const char* value);

/*
 * Set a 'value' that must not be NULL for a group by 'id' of a COSY element by 'hCosy'.
 * Return the path name as UTF8 encoded string on success, else NULL on failure.
 */
const char* cosySetGroupValue(COSY_H hCosy, const char* id, const char* value);

/*
 * Set a property value by 'pValue' and 'valueSize', which 'iecType' is specified according
 * to the convention table below, for a group by 'id' of a COSY element by 'hCosy'.
 * Return true on success, else false on failure.
 *
 * In case of 'id' represents a path to a property, like id:= "g1/g2/g3/property", all
 * parent groups will be created on demand.
 *
 * Any property that does not exist will be created, else its value will updated only in case of
 * the 'iecType' matches the existing property's type.
 *
 * Convention:
 * According to the mapping table the 'pValue' is interpreted differently. For IEC data types
 * (see iecType.h) the input parameter 'valueSize' is optional. It is used for iecType="BLOB" only.
 * Note, that the mapping convention has an impact on 'cosyGetPropertyValue' too.
 *
 * pValue       |   valueSize   |   iecType
 * -------------|---------------|-----------
 * uint32_t     |      -        |   BOOL, SINT, INT, DINT, USINT, UINT, UDINT, BYTE, WORD, DWORD
 * const char*  |      -        |   REAL, LREAL, STRING, TIME, DATE, DATE_AND_TIME, TIME_OF_DAY
 * ----------------------------------------------------------------------------------------------
 * void*        |   N bytes     |   BLOB
 *
 * Unsupported IEC data types (see iecType.h):
 * ULINT, LWORD, WSTRING, OCTET, LINT
 */
bool cosySetProperty(COSY_H hCosy, const char* id, const char* iecType, const void* pValue, size_t valueSize);

/*
 * Delete a group or property by its 'id' of a COSY element by 'hCosy'. 'timeoutUsec' is used to specify the
 * timeout [Usec] that the cleanup process is allowed to be blocked by a competitive process operating on an
 * open element. Use COSY_TIMEOUT_NO_WAIT, COSY_TIMEOUT_WAIT_FOREVER or any numeric value to regulate the timeout.
 * Return true on success, else false on failure.
 */
bool cosyDeleteMember(COSY_H hCosy, const char* id, uint32_t timeoutUsec);

/*
 * Set the 'version' of a COSY element by 'hCosy'.
 * Return true on success, false on failure.
 */
bool cosySetElementVersion(COSY_H hCosy, const char* version);

#if AR_CORE
#include <private/cosyWriteApiP.h>
#endif

#ifdef __cplusplus
}
#endif

#endif
```

#### moApi.h
```c
/* Funktionen zum Zugriff auf B&R-Module.
 *
 * Aufbau von B&R-Modulen siehe:
 * http://bratgrazpdc1/Technical%20Info/DescrBrModule/index.htm
 * bzw. ssmodul.doc
 */

#ifndef _MO_API_H_
#define _MO_API_H_

#include <rtkTypes.h>
#include <moduleTypes.h>
#include <moduleName.h>
#include <nvMemoryTypes.h>
#include <arexport.h>

#ifdef __cplusplus
extern "C" {
#endif

typedef struct BRModul_TabFS* MOHANDLE;

/* Die Iterationsfunktion liefert das Handle des ersten B&R-Modul-Objekts in der Verwaltung der B&R-Module.
 * Returns: Handle des ersten B&R-Moduls, oder NULL falls es kein B&R-Modul gibt. */
MOHANDLE moGetFirst();

/* Die Iterationsfunktion liefert das Handle des nachfolgenden B&R-Modul des mit 'hMo' spezifizierten Vorgaengers in
 * der Verwaltung der B&R-Module.
 * Returns: Handle des naechsten B&R-Moduls, oder NULL falls es kein weiteres Modul gibt. */
MOHANDLE moGetNext(MOHANDLE hMo);

/* Die Funktion sucht ein B&R-Modul ueber den Namen 'moduleName' und ermittelt das Handle des B&R-Modul-Objekts.
 * Es kann der vollqualifizierte Modulname <Scopename::B&R-Modulname> zur Suche von B&R-Modulen im Scope von
 * "AppModulen", oder der einfache B&R-Modulname <B&R-Modulname> zur Suche im "Default-Scope" angegeben werden.
 * Returns: Handle des per Namen gesuchten B&R-Moduls, oder NULL falls das B&R-Modul nicht gefunden wurde. */
MOHANDLE moFindByName(const char* moduleName);

/* Die Funktion ermittelt den Identifier fuer die DataObj-Library fuer das mit 'hMo' spezifizierte B&R-Modul.
 * Returns: Identifier fuer DataObj-Library, oder 0 falls das Modul nicht gefunden wurde. */
AR_NOT_RECOMMENDED ULONG moHandleToDataObjId(MOHANDLE hMo);

/* Die Funktion ermmittelt das Handle des B&R-Modul-Objekts fuer das mit 'id' (DataObj-Library-Modul-Identifier)
 * spezifizierte B&R-Modul.
 * Returns: Handle des B&R-Moduls, oder NULL falls das B&R-Modul nicht gefunden wurde. */
AR_NOT_RECOMMENDED MOHANDLE moDataObjIdToHandle(ULONG id);

/* Die Funktion ermittelt den Namen des ueber 'hMo' spezifizierten B&R-Moduls.
 * Der Name wird in den uebergebenen Puffer 'nameBuffer' mit maximaler Laenge 'bufferSize' kopiert.
 * Ist der Puffer zu klein, wird der Name abgeschnitten und 0-terminiert (kein Fehler!).
 * Falls das Modul Teil eines "AppModuls" ist, wird der vollqualifizierte Modulname <Scopename::B&R-Modulname>
 * ermittelt, ansonsten der einfache B&R-Modulname <B&R-Modulname>.
 * Returns: Zeiger auf uebergebenen Puffer 'nameBuffer', oder NULL im Fehlerfall. */
const char* moGetName(MOHANDLE hMo, char* nameBuffer, int bufferSize);

/* Die Funktion ermittelt eine Referenz auf den Namen des ueber 'hMo' spezifizierten B&R-Moduls.
 * Die Referenz ist nur solange gueltig, solange das B&R-Modul existiert.
 * Falls das Modul Teil eines "AppModuls" ist, wird der vollqualifizierte Modulname <Scopename::B&R-Modulname>
 * ermittelt, ansonsten der einfache B&R-Modulname <B&R-Modulname>.
 * Returns: Referenz auf den B&R-Modulnamen, oder NULL im Fehlerfall. */
const char* moGetNameRef(MOHANDLE hMo);

/* Die Funktion ermittelt den Zeiger auf das Abbild des durch 'hMo' spezifizierten B&R-Moduls im DRAM.
 * Ein Return-Wert der Funktion ungleich NULL ist das Kennzeichen fuer ein geladenes B&R-Modul!
 * Returns: Zeiger auf das Abbild des B&R-Moduls im DRAM, oder NULL fuer ein nicht geladenes B&R-Modul. */
BYTE* moGetModulePtr(MOHANDLE hMo);

/* Die Funtion ermittelt die Laenge des durch 'hMo' spezifizierten B&R-Moduls in Bytes.
 * Returns: Laenge des B&R-Moduls in Bytes, oder 0 im Fehlerfall. */
ULONG moGetSize(MOHANDLE hMo);

/* Die Funktion ermittelt den Typ des durch 'hMo' spezifizierten B&R-Moduls.
 * Returns: Modultyp BRMTYP_* oder BRMTYP_INVALID im Fehlerfall (siehe modulTypes.h). */
BYTE moGetType(MOHANDLE hMo);

/* Die Funktion ermittelt den Typ des Speichers in dem das durch 'hMo' spezifizierte B&R-Modul gespeichert ist.
 * Returns: Speichertyp MEMTYP_* oder MEMTYP_INVALID im Fehlerfall (siehe nvMemoryTypes.h). */
BYTE moGetMemType(MOHANDLE hMo);

/* Die Funktion ermittelt die Version des mit 'hMo' spezifizierten B&R-Moduls.
 * Returns: B&R-Modul-Version, oder 0xff im Fehlerfall. */
BYTE moGetVersion(MOHANDLE hMo);

/* Die Funktion ermittelt die Revision des mit 'hMo' spezifizierten B&R-Moduls.
 * Returns: B&R-Modul-Revision, oder 0xff im Fehlerfall. */
BYTE moGetRevision(MOHANDLE hMo);

/* Mit Aufruf dieser Funktion wird das Abbild des durch 'hMo' spezifizierten B&R-Moduls im DRAM erzeugt.
 * Die Checksumme des B&R-Moduls wird dabei geprueft.
 * Returns: Zeiger auf das Abbild des B&R-Moduls im DRAM, oder NULL im Fehlerfall (Checksummen-Fehler oder
 * keine/zuwenig Ressourcen stehen zur Verfuegung). */
BYTE* moLoadImage(MOHANDLE hMo);

/* Mit Aufruf dieser Funktion wird explizit der Zugriff das mit 'hMo' spezifizierte B&R-Modul signalisiert.
 * Es wird sichergestellt, dass das Handle bis zum Aufruf von moDetach gueltig ist. Ein mehrfaches moAttach ist
 * moeglich. Fuer jeden Aufruf von moAttach muss ein Aufruf von moDetach folgen.
 * Returns: TRUE, wenn ein B&R-Modul-Objekt erfolgreich "attached" wurde, sonst FALSE */
BOOLEAN moAttach(MOHANDLE hMo);
AR_DEPRECATED BOOLEAN MO_Attach(MOHANDLE hMo); /* use moAttach instead*/

/* Mit Aufruf dieser Funktion wird die Beendigung des Zugriffs auf das mit 'hMo' spezifizierte B&R-Modul signalisiert.
 */
void moDetach(MOHANDLE hMo);
AR_DEPRECATED void MO_Detach(MOHANDLE hMo); /* use moDetach instead*/

/* Die Funktion ermittelt den Offset in Bytes zur Basisadresse des durch 'hMo' spezifizierten B&R-Modul.
 * Der Offset errechnet sich aus dem (Start-)Offset der mit 'sectionIndex' adressierten B&R-Modul-Section plus dem im
 * Parameter 'sectionOffset' uebergebenen Wert.
 * Ueber den Output-Paramert 'sectionSize' (Uebergabe von NULL erlaubt) wird die Laenge der mit 'sectionIndex'
 * spezifizierten Section zurueckgegeben.
 * Returns: Den berechneten Moduloffset, bestehend auf errechnetem Offset der Section und dem uebergebenen
 * Offset innerhalb der Section, oder 0xffffffff im Fehlerfall. */
ULONG moOffset(MOHANDLE hMo, BYTE sectionIndex, ULONG sectionOffset, ULONG* sectioncSize);

/* Die Funktion liest bis zu 'nBytes' Bytes in den Puffer 'buffer' aus dem durch 'hMo' spezifizierten B&R-Modul ab dem
 * angegebenen Offset 'offset' in Bytes.
 * Der Offset in das B&R-Modul kann ueber die Funktion moOffset() berechnet werden.
 * Returns: Anzahl der erfolgreich gelesenen Bytes, oder -1 im Fehlerfall. Die Anzahl der gelesenen Bytes kann kleiner
 * sein als 'nBytes', wenn das Ende des B&R-Moduls erreicht wird. */
int moReadS(MOHANDLE hMo, BYTE* buffer, ULONG offset, ULONG nBytes);

/* Werte fuer den Parameter 'options' der Funktion moReadSEx() */
#define MO_READ_DEFAULT 0
#define MO_READ_FROM_DRAM 1
#define MO_READ_FROM_NVMEM 2

/* Die Funktion liest bis zu 'nBytes' Bytes in den Puffer 'buffer' aus dem durch 'hMo' spezifizierten B&R-Modul ab dem
 * angegebenen Offset 'offset' in Bytes.
 * Der Offset in das B&R-Modul kann ueber die Funktion moOffset() berechnet werden.
 * Mit dem Parameter 'options' kann bestimmt werden, ob der Zugriff auf das Original-Modul im NV-Speicher, oder auf die
 * Kopie im DRAM (Abbild) erfolgt.
 * 		MO_READ_DEFAULT			Zugriff auf die Kopie des B&R-Moduls im DRAM, wenn das B&R-Modul geladen ist, ansonsten
 * 								Zugriff auf das B&R-Modul im NV-Speicher; Verhalten wie moReadS()
 * 		MO_READ_FROM_DRAM		Zugriff auf die Kopie des B&R-Moduls im DRAM; Fehler bei nicht geladenen B&R-Modulen
 * 		MO_READ_FROM_NVMEM		Zugriff auf das B&R-Modul im NV-Speicher; Fehler bei B&R-Modulen ohne NV-Ablage
 * Returns: Anzahl der erfolgreich gelesenen Bytes, oder -1 im Fehlerfall. Die Anzahl der gelesenen Bytes kann kleiner
 * sein als 'nBytes', wenn das Ende des B&R-Moduls erreicht wird. */
int moReadSEx(MOHANDLE hMo, BYTE* buffer, ULONG offset, ULONG nBytes, ULONG options);

/* Die Funktion schreibt 'nBytes' Bytes vom Puffer 'buffer' in das durch 'hMo' spezifizierte B&R-Modul ab dem
 * angegebenen Offset 'offset'. Der Offset in das B&R-Modul kann ueber die Funktion moOffset() berechnet werden.
 * Returns: Anzahl der erfolgreich geschriebenen Bytes, oder -1 im Fehlerfall. Da ein B&R-Modul nicht wachsen kann, wird
 * ein Fehler zurueckgegeben, wenn der die zu schreibenden Daten nicht im B&R-Modul Platz haben. */
int moWriteS(MOHANDLE hMo, BYTE* buffer, ULONG offset, ULONG nBytes);

/* Diese Funktion ermittelt assoziierte Objekte zu dem durch 'hMo' spezifizierten B&R-Modul.
 * Ist das B&R-Modul ein "Anwenderprogramm" (BRMTYP_SPSTASK/0x11) wird ein Handle vom Typ CYPHANDE zurueckgegeben.
 * Ist das B&R-Modul ein "Systemmodul" (BRMTYP_SYSTASK/0x12) wird ein Handle vom Typ NCYCHANDLE zurueckgegeben.
 * Fuer alle anderen B&R-Modultypen oder im Fehlerfall (MOHANDLE ist ungueltig) wird NULL zurueckgegeben. */
AR_NOT_RECOMMENDED LPVOID moGetObjectHandle(MOHANDLE hMo);

/* Diese Funktion ermittelt das Aenderungsdatum und -uhrzeit des durch 'hMo' spezifizierten B&R-Moduls.
 * Ueber den Output-Paramert 'time' wird das Aenderungsdatum und -uhrzeit zurueckgegeben.
 * Returns: TRUE, wenn Aenderungsdatum und -uhrzeit ermittelt werden konnten, sonst FALSE */
BOOLEAN moGetMTime(MOHANDLE hMo, RTK_RTC* time);

#if AR_CORE
#include <private/moApiP.h>
#endif

#ifdef __cplusplus
}
#endif

#endif
```

#### moduleName.h
```c
/* B&R-Modulename constants
 */

#ifndef _MODULE_NAME_H_
#define _MODULE_NAME_H_

/* identifier of default-scope */
#define DEFAULT_SCOPE_NAME ""

/* delimiter */
#define DELIMITER_SCOPE "::"
#define SCOPE_DELIMITER_LEN 2 /* scope-delimiter "::" */
#define DELIMITER_MODULE ":"
#define MODULE_DELIMITER_LEN 1 /* module-delimiter ":" */

/* name-length defines for B&R-modules */
#define MAX_SCOPE_NAME_LEN 20  /* scopename */
#define MAX_MODULE_NAME_LEN 10 /* B&R-modulename */
                               /* If max. B&R-module name-length is changed, following defines have to be changed too:
                                * - NVM_NAMELEN in NvMemory.h
                                * - ARPROF_MAX_NAME in ArProfilerP.h
                                */

#define MAX_FQ_MODULE_NAME_LEN (MAX_SCOPE_NAME_LEN + SCOPE_DELIMITER_LEN + MAX_MODULE_NAME_LEN)
/* fully qualified -> "<scopename>::<B&R-modulename>" */

/* used by different *GetName() functions (mo-API, cyp-API, ...), parameter 'ulOptions' */
#define NAME_FQ 0      /* get fully qualified modulename <Scopename::B&R-Modulename> */
#define NAME_SCOPE 1   /* get scopename only */
#define NAME_MODULE 2  /* get modulename only (scope is stripped) */
#define NAME_DEFAULT 3 /* call in default scope behaves like option MO_NAME_MODULE, otherwise like option MO_NAME_FQ*/

#endif
```

#### moduleTypes.h
```c
/*  B&R-Moduletypes and groups */

#ifndef _MODULE_TYPES_H_
#define _MODULE_TYPES_H_

/* Modulegroups */
#define BRMGRP_MASK 0xF0
#define IS_BRMGRP(modType, group) ((modType & BRMGRP_MASK) == group)
#define GET_BRMGRP(type) ((type)&0xF0)

#define BRMTYP_INVALID 			255

/* Moduletypes */
/* clang-format off */
#define BRMGRP_VW			(0 << 4)	/* Gruppe Verwaltungsmodule */
/*#define BRMTYP_RPSSW_UPDATE	0*/		/* 0x00 RPSSW-Update */
#define BRMTYP_TRSFM			1		/* 0x01 Transfermodul, ehemals BRMTYP_INHVZ = Inhaltsverzeichnis */
/*#define BRMTYP_INHVF			2*/		/* 0x02 InhVZ Fortsetzung */
/*#define BRMTYP_MEMEX			3*/		/* 0x03 Speicherextension */
/*#define BRMTYP_HWD			4*/		/* 0x04 Hardwarebeschreibung (nur fuer SG4)*/
/*#define BRMTYP_START			7*/		/* 0x07 Bootmodul */

#define BRMGRP_TASK			(1 << 4)	/* Gruppe Taskmodule */
#define BRMTYP_SPSTASK			17		/* 0x11 SPSTask Modul */
#define BRMTYP_SYSTASK			18		/* 0x12 Systemtask Modul */
/*#define BRMTYP_USERTASK		19*/	/* 0x13 Usertask Modul */
/*#define BRMTYP_SSTASK			20*/	/* 0x14 SS Task Modul */
/*#define BRMTYP_IRQTASK		21*/	/* 0x15 Interrupttask Modul */
#define BRMTYP_EXCTASK			22		/* 0x16 Exceptiontask Modul */
/*#define BRMTYP_STARTUP		31*/	/* 0x1F Modultyp des Startup-Moduls */

/*#define BRMGRP_LIB		(2 << 4)*/	/* Gruppe Library-/Trap-Module */
/*#define BRMTYP_UPLIB			33*/	/* 0x21 FUB/UP AVT Lib */
/*#define BRMTYP_SYSLIB			34*/	/* 0x22 SystemSW Lib */
/*#define BRMTYP_HWLIB			35*/	/* 0x23 Hardwaretrap Lib */
/*#define BRMTYP_KOMLIB			36*/	/* 0x24 Kommuni(ALI) Lib */
/*#define BRMTYP_MATHLIB		37*/	/* 0x25 Mathematik Lib */
/*#define BRMTYP_LIB			38*/	/* 0x26 irgendeine Lib */
/*#define BRMTYP_INSTLIB		39*/	/* 0x27 Insttrap */
/*#define BRMTYP_ADDLIB			40*/	/* 0x28 Erweiterungstrap */

#define BRMGRP_IO			(3 << 4)	/* Gruppe IO-Module */
/*#define BRMTYP_IO				49*/	/* 0x31 IO-Modul SchTab */
#define BRMTYP_IOMAP			50		/* 0x32 IO-Map (nur fuer SG4) */

#define BRMGRP_TAB			(4 << 4)	/* Gruppe Tabellenmodule */
#define BRMTYP_BRDATA			65		/* 0x41 B&R Datenmodul */
/*#define BRMTYP_SDMDATA		66*/	/* 0x42 System Diagnostics Datenmodul */
#define BRMTYP_CONTAINER		67		/* 0x43 Containermodul */
#define BRMTYP_SAFETY_APP		68		/* 0x44 Safety Application (als Binaerstrom in der Datensection) */
#define BRMTYP_NC_TREIBER		69		/* 0x45 */
#define BRMTYP_NC_DATA			70		/* 0x46 entspricht BRMTYP_BRNCDATA von Motion */
#define	BRMTYP_SAFETY_CONFIG	71		/* 0x47 Safety Konfigurationsdaten */
/*#define BRMTYP_XTRACE_DEF		73*/	/* 0x49 Trace Definition fuer "Oszi-Module" */
/*#define BRMTYP_XTRACE_DATA	74*/	/* 0x4A Trace Daten fuer "Oszi-Module" */
#define BRMTYP_PROFILE_DEF		75		/* 0x4B Profile Definition */
#define BRMTYP_PROFILE_DATA		76		/* 0x4C Profile Daten */
#define BRMTYP_TRACER_DEF		77		/* 0x4D Tracer Definition */
#define BRMTYP_TRACER_DATA		78		/* 0x4E Tracer Daten */
#define BRMTYP_NC_UPDATE		79		/* 0x4F */

#define BRMGRP_RING			(5 << 4)	/* Gruppe Ringpuffermodule */
/*#define BRMTYP_HIST			81*/	/* 0x51 Historymodul */
#define BRMTYP_ERROR			82		/* 0x52 Errormodul */
#define BRMTYP_LOGGER			83		/* 0x53 Loggermodul */

/*#define BRMGRP_COPY		(6 << 4)*/	/* Gruppe Copy-Module */
/*#define BRMTYP_NOC			97*/	/* 0x61 NW Output Copymodul */

/*#define BRMGRP_PA			(7 << 4)*/	/* Gruppe Prozessabbildmodule */
/*#define BRMTYP_MERKER			113*/	/* 0x71 PA Merkerabbild */
/*#define BRMTYP_TKLOC			114*/	/* 0x72 PA tasklokaler Sp */

#define BRMGRP_CONF			(8 << 4)	/* Konfigurationsmodule */
#define BRMTYP_CFGSPS			129		/* 0x81 SPS Konfiguration */
/*#define BRMTYP_CFGKOM			130*/	/* 0x82 KOM Konfiguration */
/*#define BRMTYP_CFGPP			131*/	/* 0x83 PeriProz Konf */
#define BRMTYP_CFGIO			132		/* 0x84 IO Konfiguration (arconfig.br - nur fuer SG4) */
/*#define BRMTYP_CFGOPC			133*/	/* 0x85 OPC Konfiguration (asopc - nur fuer SG4) */
#define BRMTYP_CFGOPCUA			134		/* 0x86 OPC-UA Konfiguration */
#define BRMTYP_CFGRRAD			135		/* 0x87 Redundanz Relevante Anwenderdaten */
#define BRMTYP_CFGXML			136		/* 0x88 XML-basiertes Konfigurationsmodul (GSA) */
#define BRMTYP_CFGXMLS			137		/* 0x89 XML-basiertes Konfigurationsmodul (GSA) - Persistente Sicherung */
/*#define BRMTYP_CFGTRACE		138*/	/* 0x8A Zentraler Aufzeichnungsmechanismus Konfiguration (GSA) */
/*#define BRMTYP_CFG			143*/	/* 0x8F beliebiges Konfigurationsmodul */

/*#define BRMGRP_EXC_IRQ	(9 << 4)*/	/* Exception-/IRQ-Module */
/*#define BRMTYP_EXCEP			145*/	/* 0x91 Exceptionmodul */
/*#define BRMTYP_IRQ			146*/	/* 0x92 IRQ Modul */

/*#define BRMGRP_DEVICE		(0x0a << 4)*/	/* Gruppe Device-Driver-Modul */
/*#define BRMTYP_DEVICE			161*/	/* 0xA1 Devicedrivermodul */

/*#define BRMGRP_TAB_NG		(0x0b << 4)*/	/* Gruppe Tabellenmodule (Fortsetzung von BRMGRP_TAB) */
/*#define BRMTYP_CAPTRACE		177*/	/* 0xB1 Zentraler Aufzeichnungsmechanismus Capture (GSA) */

/*#define BRMGRP_UP			(0x0c << 4)*/	/* Gruppe UP-Module */
/*#define BRMTYP_UP				193*/	/* 0xC1 Unterprogrammmodul */

#define BRMGRP_DB			(0x0d << 4)	/* Gruppe Datenbankmodule */
/*define BRMTYP_SQLITE0			208*/	/* 0xD0*/
#define BRMTYP_SQLITE_TEXT		209 	/* 0xD1 Textsystem SQLite DBs	*/
/*define BRMTYP_SQLITE2			210*/	/* 0xD2 */
#define BRMTYP_SQLITE_TEXT_EXT	211		/* 0xD3 Nachladbare SQLite Textsystem DBs */

/*#define BRMGRP_EXE		(0x0e << 4)*/	/* Gruppe EXE-Module */
/*#define BRMTYP_EXE			224*/	/* 0xE0 beliebiges EXE Modul */
/*#define BRMTYP_PR				237*/	/* 0xED Modultyp des pROBE-Moduls*/
/*#define BRMTYP_PI				238*/	/* 0xEE Modultyp des pROBE-IO */
/*#define BRMTYP_OS				239*/	/* 0xEF Betriebssystem EXE */

/*#define BRMGRP_DATA		(0x0f << 4)*/	/* Gruppe Datenmodule */
/*#define BRMTYP_DATA			240*/	/* 0xF0 beliebiges Daten Modul */
/* clang-format on */

#endif
```

#### nvMemoryTypes.h
```c
/* Non Volatile (NV) Memory Types */

#ifndef _NV_MEMORY_TYPES_H_
#define _NV_MEMORY_TYPES_H_

/* clang-format off */
#define	MEMTYP_SYSTEM_FLASH			0		/* System ROM */
#define	MEMTYP_SYSTEM_RAM			1		/* obsolet, only used by MEM_gettyp() */
#define	MEMTYP_USER_FLASH			2		/* User ROM */
#define	MEMTYP_USER_RAM				3		/* User RAM */
#define	MEMTYP_COPY_RAM				0x41	/* Heap/DRAM */
#define	MEMTYP_SYSTEM_FLASH_BURN	0xEE	/* System ROM, only used by online communication */
#define	MEMTYP_PERMANENT_MEM		0xF0	/* system internal permanent memory */
#define	MEMTYP_SYSTEM_INTERNAL		0xF1	/* system internal memory for simulated B&R-Modules */
#define	MEMTYP_REMANENT_MEM			0xF2	/* memory for VAR_RETAIN (remanent + permanent PVs) */
#define	MEMTYP_ARREGNV_MEM			0xF3	/* memory for non volatile system configuration */
#define	MEMTYP_TRSF					0xF4	/* memory for transfer module */

#define	MEMTYP_INVALID				0xFF	/* memory not supported */

#endif
```

### Program Logical/HMI

#### Variables.var
```iecst
VAR
	TON_Reset : TON;
END_VAR
```

#### Main.st
```iecst
PROGRAM _INIT
	(* Insert code here *)

END_PROGRAM

PROGRAM _CYCLIC
	(* Insert code here *)
	(*
	IF gHMI.General.PlayButton THEN
		IF MAIN_DISABLED = MainState THEN
			gMain.Cmd.Power := TRUE;
		END_IF;
	ELSIF gHMI.General.StopButton THEN
		gMain.Cmd.Power := FALSE;
	ELSIF gHMI.General.ResetButton THEN
		IF MainState = MAIN_ERROR THEN
			gMain.Cmd.ErrorReset := TRUE;
		END_IF;
	END_IF;
	*)

	IF gHMI.Game.NewGame OR gHMI.Game.ExitGame THEN
		brsmemset(ADR(gHMI.Game),0,SIZEOF(gHMI.Game));
	END_IF;

	TON_Reset.IN := gHMI.General.ResetPLC;
	TON_Reset.PT := TIME#5s;
	TON_Reset;

	IF TON_Reset.Q THEN
		SYSreset(1,1);
	END_IF;
END_PROGRAM

PROGRAM _EXIT
	(* Insert code here *)

END_PROGRAM
```

### Types.typ
```iecst
TYPE
	Acp6DCmdType : 	STRUCT
		PowerOn : BOOL;
		PowerOff : BOOL;
		Init : BOOL;
		StartProcess : BOOL;
		StopProcess : BOOL;
		Stop : BOOL;
		gameProgramDeleteShuttle : BOOL;
		Reset : BOOL;
	END_STRUCT;
	Acp6DCtrlType : 	STRUCT
		Cmd : Acp6DCmdType;
		Status : Acp6DStatusType;
		Par : Acp6DParType;
	END_STRUCT;
	Acp6DParType : 	STRUCT
		Acceleration : REAL := 10;
		Velocity : REAL := 2;
		modeSelectorOld : driveModes;
		modeSelector : driveModes;
		rotationVelocity : REAL := 30;
		rotationAcceleration : REAL := 30;
	END_STRUCT;
	Acp6DStatusType : 	STRUCT
		Error : BOOL;
		ErrorID : DINT;
		Ready : BOOL;
		PowerOn : BOOL;
		ReadyToPowerOn : BOOL;
		SegmentInfo : ARRAY[0..NUM_SEGMENTS]OF segmentInfoType;
		ShuttleInfo : ARRAY[0..NUM_SHUTTLES]OF ShuttleInfoType;
		ShuttleInfoVis : ARRAY[0..NUM_SHUTTLES]OF ShuttleInfoType;
		currentNumShuttles : UINT;
	END_STRUCT;
	box_typ : 	STRUCT
		smallBox : BOOL;
		bottle : BOOL;
		bigBox : BOOL;
	END_STRUCT;
	driveModes :
		(
		none := 0, (*bootup*)
		vision := 1,
		weight := 2,
		linkMovement := 3,
		gameProgram := 4,
		demoProgram := 5,
		shuttleToConveyor := 6,
		workstationMovement := 8,
		conveyorStationMovement := 9,
		dialGauge := 7,
		danfossMode := 10,
		sunMovement := 11,
		flaskProgram := 12,
		boxProgram := 13,
		rotationProgram := 14,
		steelSheet := 15,
		teachProgramEnum := 16,
		trakModeEnum := 17,
		rotationSyncEnum := 18
		);
	segmentInfoType : 	STRUCT
		ID : UINT;
		segmentRef : Mc6DSegmentType;
	END_STRUCT;
	ShuttleInfoType : 	STRUCT
		ID : UINT;
		State : McAcp6DShStateEnum;
		Force : McAcp6DShForceType;
		Position : McAcp6DShPositionType;
		inUse : BOOL; (*DryStation Bool*)
		lastgPath : DINT := 100;
		shuttleRef : Mc6DShuttleType;
	END_STRUCT;
	shuttleStartup_typ : 	STRUCT
		initYPos : REAL;
		initXPos : REAL;
		nextStationSelector : STRING[80] := '0';
		initZPos : REAL;
		initRxPos : REAL;
		initRyPos : REAL;
		initRzPos : REAL;
	END_STRUCT;
	workStation_cmd_typ : 	STRUCT
		dummy : USINT;
	END_STRUCT;
	workStation_par_typ : 	STRUCT
		landBeforeProcess : BOOL; (*TRUE = yes*)
		yLocation : REAL;
		xLocation : REAL;
		tempShuttleID : USINT;
		processTime : REAL;
		pathRouting : USINT := 0; (*0 Diagonal, 1 First X then Y, 2 First Y then X*)
		nextStationSelector : STRING[80];
		ArcMovement : BOOL;
		internalCounter : USINT;
		tempCounter : USINT;
	END_STRUCT;
	workStation_status_typ : 	STRUCT
		componentName : STRING[80];
		active : BOOL;
		oneshot : BOOL;
	END_STRUCT;
	workStation_typ : 	STRUCT
		par : workStation_par_typ;
		status : workStation_status_typ;
		cmd : workStation_cmd_typ;
		cm : brdkCM;
		MC_BR_RotaryMotionSpin_Acp6D_0 : MC_BR_RotaryMotionSpin_Acp6D;
		MC_BR_RotaryMotion_Acp6D_0 : MC_BR_RotaryMotion_Acp6D;
		MC_BR_MoveInPlane_Acp6D_0 : MC_BR_MoveInPlane_Acp6D;
		MC_BR_ShLevitation_Acp6D_0 : MC_BR_ShLevitation_Acp6D;
		TON_0 : TON;
		workstationSwitcher : BOOL;
		MC_BR_MoveArc_Acp6D_0 : MC_BR_MoveArc_Acp6D;
		MC_BR_Move6D_Acp6D_0 : MC_BR_Move6D_Acp6D;
		MC_BR_MoveShortAxis_Acp6D_0 : MC_BR_MoveShortAxis_Acp6D;
	END_STRUCT;
END_TYPE
```

### Variables.var
```iecst
VAR
	gWorkStations : {REDUND_UNREPLICABLE} ARRAY[0..NR_OF_WORKSTATIONS] OF workStation_typ;
	shuttleStartupInfo : ARRAY[0..NUM_SHUTTLES] OF shuttleStartup_typ;
	cmdBoxProgram : box_typ;
	gAcp6DCtrl : Acp6DCtrlType;
	ShuttleYPos_m : LREAL;
END_VAR
(*Constants*)
VAR CONSTANT
	NUM_SEGMENTS : USINT := 1; (*2[0..1]*)
	NUM_SHUTTLES : USINT := 3; (*4[0..3]*)
	NR_OF_WORKSTATIONS : USINT := 3; (*4[0..3]*)
END_VAR
```

### Program Logical/Modules/Acopos6D/Acopos6D (IEC)

#### Main.st - Init, cyclic, exit code
```iecst
PROGRAM _INIT
	em.setup.name := 'Acopos6D';
	em.setup.parent.name := 'main';
	em();

	MC_BR_AsmGetInfo_Acp6D_0.Assembly			:= ADR(gAssembly6D_1);
	MC_BR_AsmGetSegment_Acp6D_0.Assembly		:= ADR(gAssembly6D_1);
	MC_BR_AsmGetShuttle_Acp6D_0.Assembly 		:= ADR(gAssembly6D_1);
	MC_BR_AsmReadStatus_Acp6D_0.Assembly 		:= ADR(gAssembly6D_1);
	MC_BR_AsmPowerOn_Acp6D_0.Assembly			:= ADR(gAssembly6D_1);
	MC_BR_AsmPowerOff_Acp6D_0.Assembly			:= ADR(gAssembly6D_1);
	MC_BR_AsmStop_Acp6D_0.Assembly				:= ADR(gAssembly6D_1);
	MC_BR_MoveInPlaneAsync_Acp6D_0.Assembly		:= ADR(gAssembly6D_1);
	MC_BR_ShGroupCreate_Acp6D_0.Assembly 		:= ADR(gAssembly6D_1);
	MC_BR_ShGroupCreate_Acp6D_1.Assembly 		:= ADR(gAssembly6D_1);
	MC_BR_ShGroupCreate_Acp6D_2.Assembly 		:= ADR(gAssembly6D_1);
	MC_BR_ShGroupCreate_Acp6D_3.Assembly 		:= ADR(gAssembly6D_1);
	MC_BR_MacroCreate_Acp6D_0.Assembly			:= ADR(gAssembly6D_1);
	MC_BR_AsmLevitation_Acp6D_0.Assembly		:= ADR(gAssembly6D_1);
	MC_BR_AsmReset_Acp6D_0.Assembly 			:= ADR(gAssembly6D_1);

	MC_BR_AsmReadStatus_Acp6D_0.Enable			:= TRUE;
	//MC_BR_AsmGetInfo_Acp6D_0.Execute := TRUE;

	MC_BR_AsmReadStatus_Acp6D_0();
END_PROGRAM

PROGRAM _CYCLIC
	// Setup config parameters
	config;

	// IF 6D Controller goes into Error PackML State machine will follow
	IF MC_BR_AsmReadStatus_Acp6D_0.Valid AND MC_BR_AsmReadStatus_Acp6D_0.AssemblyErrorStop AND em.state <> STATE_ABORTED THEN
		em.cmd.abort := TRUE;
	END_IF

	CASE em.state OF
		STATE_STOPPED:
			em.description := 'Waiting for reset cmd';
			IF MC_BR_AsmReadStatus_Acp6D_0.AssemblyDisabled AND NOT MC_BR_AsmReadStatus_Acp6D_0.AssemblyErrorStop THEN
				em.cmd.sc := TRUE;
			ELSE
				em.cmd.sc := FALSE;
			END_IF

		STATE_RESETTING:
			CASE em.substate OF
				0:
					em.description := 'Reset all inputs';
					ResetInput;
					em.substate := 2;

				2:
					MC_BR_AsmGetInfo_Acp6D_0.Execute := TRUE;
					IF MC_BR_AsmGetInfo_Acp6D_0.Done THEN
						gAcp6DCtrl.Status.currentNumShuttles := MC_BR_AsmGetInfo_Acp6D_0.AssemblyInfo.NumberOfShuttles;
						localCurrentNumShuttles := gAcp6DCtrl.Status.currentNumShuttles;
						MC_BR_AsmGetInfo_Acp6D_0.Execute := FALSE;
						IF gAcp6DCtrl.Status.currentNumShuttles > 0 THEN
							em.substate := 5;
						ELSE
							em.cmd.abort := TRUE;
						END_IF
					END_IF

				5:
					em.description := 'Load shuttle IDs';
					MC_BR_AsmGetShuttle_Acp6D_0.Enable := TRUE;
					gAcp6DCtrl.Status.currentNumShuttles := MC_BR_AsmGetInfo_Acp6D_0.AssemblyInfo.NumberOfShuttles;
					IF MC_BR_AsmGetShuttle_Acp6D_0.Valid AND MC_BR_AsmGetShuttle_Acp6D_0.Busy THEN
						tempCounter := 0;
						em.substate := 6;
					END_IF

				6:
					em.description := 'copy shuttle ref';
					MC_BR_AsmGetShuttle_Acp6D_0.Next := FALSE;
					gAcp6DCtrl.Status.ShuttleInfo[MC_BR_AsmGetShuttle_Acp6D_0.AdditionalInfo.ShuttleID-1].ID := MC_BR_AsmGetShuttle_Acp6D_0.AdditionalInfo.ShuttleID;
					gAcp6DCtrl.Status.ShuttleInfo[MC_BR_AsmGetShuttle_Acp6D_0.AdditionalInfo.ShuttleID-1].shuttleRef := MC_BR_AsmGetShuttle_Acp6D_0.Shuttle;
					IF MC_BR_AsmGetShuttle_Acp6D_0.Shuttle.controlif = 0 THEN
						MC_BR_AsmGetShuttle_Acp6D_0.Enable := FALSE;
						em.cmd.abort := TRUE;
					ELSIF MC_BR_AsmGetShuttle_Acp6D_0.RemainingCount = 0 THEN
						//MC_BR_AsmGetShuttle_Acp6D_0.Enable := FALSE;
						em.substate := 10;
					ELSE
						em.substate := 7;
					END_IF

				7:
					MC_BR_AsmGetShuttle_Acp6D_0.Next := TRUE;
					em.substate := 6;

				10:
					em.description := 'Power on 6DController';
					IF MC_BR_AsmReadStatus_Acp6D_0.AssemblyReady THEN
						em.substate := 15;
					ELSE
						MC_BR_AsmPowerOn_Acp6D_0.Execute 			:= TRUE;
						IF(MC_BR_AsmPowerOn_Acp6D_0.Acknowledge AND MC_BR_AsmPowerOn_Acp6D_0.Done)THEN
							MC_BR_AsmPowerOn_Acp6D_0.Execute 		:= FALSE;
							em.substate  							:= 15;
						ELSIF(MC_BR_AsmPowerOn_Acp6D_0.Error)THEN
							MC_BR_AsmPowerOn_Acp6D_0.Execute 		:= FALSE;
							em.cmd.abort							:= TRUE;
						END_IF;
					END_IF

				15:
					em.description := 'Check Assembly Ready';
					IF MC_BR_AsmReadStatus_Acp6D_0.AssemblyReady THEN
						em.substate := 20;
						tempShuttleCnt := 0;
					ELSE
						em.substate := 10; //Sometimes AsmPowerOn dont power on the system
					END_IF

				20:
					em.description := 'Get segmentID';
					MC_BR_AsmGetSegment_Acp6D_0.Enable := TRUE;
					IF MC_BR_AsmGetSegment_Acp6D_0.Valid AND MC_BR_AsmGetSegment_Acp6D_0.Busy THEN
						tempCounter := 0;
						em.substate := 21;
					END_IF

				21:
					em.description := 'copy Segment ref';
					MC_BR_AsmGetSegment_Acp6D_0.Next := FALSE;
					gAcp6DCtrl.Status.SegmentInfo[MC_BR_AsmGetSegment_Acp6D_0.AdditionalInfo.SegmentID-1].ID := MC_BR_AsmGetSegment_Acp6D_0.AdditionalInfo.SegmentID;
					gAcp6DCtrl.Status.SegmentInfo[MC_BR_AsmGetSegment_Acp6D_0.AdditionalInfo.SegmentID-1].segmentRef := MC_BR_AsmGetSegment_Acp6D_0.Segment;
					IF MC_BR_AsmGetSegment_Acp6D_0.RemainingCount = 0 THEN
						//MC_BR_AsmGetSegment_Acp6D_0.Enable := FALSE;
						em.substate := 23;
					ELSE
						em.substate := 22;
					END_IF

				22:
					MC_BR_AsmGetSegment_Acp6D_0.Next := TRUE;
					em.substate := 21;

				23:
					em.description := 'Break all shuttles';
					MC_BR_AsmStop_Acp6D_0.Execute := TRUE;
					IF MC_BR_AsmStop_Acp6D_0.Done THEN
						MC_BR_AsmStop_Acp6D_0.Execute := FALSE;
						em.substate := 25;
					END_IF

				25:
					em.description := 'Check all shuttles states';
					IF gAcp6DCtrl.Status.ShuttleInfo[tempShuttleCnt].State = mcACP6D_SH_STATE_IDLING THEN
						tempShuttleCnt := tempShuttleCnt + 1;
						em.substate := 27;
					ELSE
						em.substate := 15;
					END_IF

				27:
					em.description := 'all shuttles checked?';
					IF tempShuttleCnt > localCurrentNumShuttles-1 THEN
						em.substate := 40;
					ELSE
						em.substate := 25;
					END_IF

				40:
					em.description := 'Check one shuttle to see if MoveInPlaceAsync is done';
					IF gAcp6DCtrl.Status.ShuttleInfo[0].State =  mcACP6D_SH_STATE_IDLING THEN
						em.substate := 90; //cant use Async when stereoType is defined
					END_IF

				90:
					shuttleGroups;
					macroCreatorAction;
					IF createShGroup = 80 AND macroCreater = 70 THEN
						em.substate := 100;
					END_IF

				100:
					MC_BR_ShGroupGetInfo_Acp6D_0.ShuttleGroup := shGroupShuttle1_2;
					MC_BR_ShGroupGetInfo_Acp6D_0.Execute := TRUE;
					em.cmd.sc := TRUE;
			END_CASE

		STATE_STARTING:
			CASE em.substate OF
				0:
					IF gAcp6DCtrl.Status.ShuttleInfo[0].State =  mcACP6D_SH_STATE_IDLING AND gAcp6DCtrl.Status.ShuttleInfo[1].State =  mcACP6D_SH_STATE_IDLING AND gAcp6DCtrl.Status.ShuttleInfo[2].State =  mcACP6D_SH_STATE_IDLING
						AND gAcp6DCtrl.Status.ShuttleInfo[3].State =  mcACP6D_SH_STATE_IDLING THEN
						em.substate := 2;
					END_IF

				2:
					em.description := 'Break all shuttles';
					MC_BR_AsmStop_Acp6D_0.Execute := TRUE;
					IF MC_BR_AsmStop_Acp6D_0.Done THEN
						MC_BR_AsmStop_Acp6D_0.Execute := FALSE;
						em.substate := 3;
					END_IF

				3:
					IF gAcp6DCtrl.Status.ShuttleInfo[0].State =  mcACP6D_SH_STATE_IDLING AND gAcp6DCtrl.Status.ShuttleInfo[1].State =  mcACP6D_SH_STATE_IDLING AND gAcp6DCtrl.Status.ShuttleInfo[2].State =  mcACP6D_SH_STATE_IDLING
						AND gAcp6DCtrl.Status.ShuttleInfo[3].State =  mcACP6D_SH_STATE_IDLING THEN
						em.substate := 5;
					END_IF

				5:
					em.description := 'Move to start pos';
					TON_watchdog.IN := FALSE; // Firmware bugfix
					TON_watchdog.PT := t#4s; // Firmware bugfix
					MC_BR_MoveInPlaneAsync_Acp6D_0.Parameters.Acceleration := gAcp6DCtrl.Par.Acceleration;
					MC_BR_MoveInPlaneAsync_Acp6D_0.Parameters.Velocity := gAcp6DCtrl.Par.Velocity;
					FOR i := 0 TO UINT_TO_USINT(localCurrentNumShuttles-1) DO
						MC_BR_MoveInPlaneAsync_Acp6D_0.Parameters.AsyncPar[i].Shuttle := ADR(gAcp6DCtrl.Status.ShuttleInfo[i].shuttleRef);
						MC_BR_MoveInPlaneAsync_Acp6D_0.Parameters.AsyncPar[i].X := shuttleStartupInfo[i].initXPos;
						MC_BR_MoveInPlaneAsync_Acp6D_0.Parameters.AsyncPar[i].Y := shuttleStartupInfo[i].initYPos;
					END_FOR
					MC_BR_MoveInPlaneAsync_Acp6D_0.Execute := TRUE;
					IF MC_BR_MoveInPlaneAsync_Acp6D_0.Done THEN
						MC_BR_MoveInPlaneAsync_Acp6D_0.Execute := FALSE;
						em.substate := 10;
					END_IF
					// Firmware bugfix - Sometimes MoveInPlaneAsync is stuck and will need a FB reset
					IF MC_BR_MoveInPlaneAsync_Acp6D_0.Busy THEN
						TON_watchdog.IN := TRUE;
						IF TON_watchdog.Q THEN
							MC_BR_MoveInPlaneAsync_Acp6D_0.Execute := FALSE;
						END_IF
					END_IF

				10:
					em.cmd.sc := TRUE;
			END_CASE

		STATE_EXECUTE:
			em.description := 'Shuttle program with selected mode is running';
			gAcp6DCtrl.Status.Ready := TRUE;
			em.cmd.sc := TRUE;

			CASE em.substate OF
				0:
					CASE gAcp6DCtrl.Par.modeSelector OF
						vision: em.substate := 1000;
						weight: em.substate := 2000;
						linkMovement: em.substate := 3000;
						gameProgram: em.substate := 4000;
						demoProgram: em.substate := 5000;
						shuttleToConveyor: em.substate := 6000;
						dialGauge: em.substate := 7000;
						workstationMovement: em.substate := 8000;
						conveyorStationMovement: em.substate := 9000;
						danfossMode: em.substate := 10000;
						sunMovement: em.substate := 11000;
						flaskProgram: em.substate := 12000;
						boxProgram: em.substate := 13000;
						rotationProgram: em.substate := 14000;
						steelSheet: em.substate := 15000;
						teachProgramEnum: em.substate := 16000;
						trakModeEnum: em.substate := 17000;
						rotationSyncEnum: em.substate := 18000;
					END_CASE

				2000..2999:
					enableButtons := FALSE;
					em.cmd.sc := FALSE;
					em.description := 'Weight Program';
					IF controlLight.weightProgram THEN
						lightValue := 6;
					END_IF

					FOR i := 0 TO NUM_SHUTTLES DO
						pShuttle ACCESS ADR(gShuttles[i]);
						cm ACCESS ADR (gShuttles[i].cm);
						pShuttle.cm.setup.parent.name := 'main';
						pShuttle.cm.setup.nameIdx := i;
						pShuttle.par.shuttleID := i;

						//Chosen action pr shuttle
						CASE i OF
							0:weightProgram;
							3:MovementRx;
							2:MovementRy;
							1:MovementZ;
						END_CASE
					END_FOR
					em.cmd.sc := TRUE;

				3000..3999:
						em.description := 'linkMovement Program';
						IF controlLight.linkProgram THEN
							lightValue := 3;
						END_IF

						linkMovementProgram;

				5000..5999:
					em.description := 'Demo program';
					IF controlLight.demoProgram THEN
						lightValue := 5;
					END_IF

					demoProgramTask;

				7000:
					em.description := 'dialGauge Program';
					IF controlLight.shuttlePrecision THEN
						lightValue := 4;
					END_IF

					FOR i := 0 TO NUM_SHUTTLES DO
						pShuttle ACCESS ADR(gShuttles[i]);
						cm ACCESS ADR (gShuttles[i].cm);
						pShuttle.cm.setup.parent.name := 'main';
						pShuttle.cm.setup.nameIdx := i;
						pShuttle.par.shuttleID := i;

						//Chosen action pr shuttle
						CASE i OF
							0:MovementRy;
							1:MovementZ;
							2:MovementRx;
							3:BasicMoveDialGauge;
						END_CASE
					END_FOR
					em.cmd.sc := TRUE;

				8000..8002:
				workStationSetup;

				8003..8999:
					workStationSetup;
					em.description := 'intelligentMovement';
					IF controlLight.intelligentMovementProgram THEN
						lightValue := 7;
					END_IF
						FOR i := 0 TO NR_OF_WORKSTATIONS DO
							pWorkStations ACCESS ADR (gWorkStations[i]);
						cm ACCESS ADR (gWorkStations[i].cm);
						pWorkStations.cm.setup.parent.name := 'main';
						//pShuttle.cm.setup.nameIdx := i;
						workStationMovement;
						END_FOR

				9000..9002:
					conveyorStationSetup;

				9003..9999:
					em.description := 'ConveyorMovement';
					conveyorStationSetup;
					FOR i := 0 TO NR_OF_WORKSTATIONS DO
						pWorkStations ACCESS ADR (gWorkStations[i]);
						cm ACCESS ADR (gWorkStations[i].cm);
						pWorkStations.cm.setup.parent.name := 'main';
						//pShuttle.cm.setup.nameIdx := i;
						conveyourStationMovement;
					END_FOR

				10000..10999:
						em.description := 'Danfoss mode';
						danfossAction;
						FOR i := 0 TO NR_OF_WORKSTATIONS DO
							pWorkStations ACCESS ADR (gWorkStations[i]);
							cm ACCESS ADR (gWorkStations[i].cm);
							pWorkStations.cm.setup.parent.name := 'main';
							//pShuttle.cm.setup.nameIdx := i;
							DanFossWork;
						END_FOR

				12000..12019:
						em.description := 'Flask Program';
						flaskProgramTask;

				12020..12999:
						em.description := 'Flask Program';
						flaskProgramTask;
						FOR i := 0 TO NUM_SHUTTLES DO
							pShuttle ACCESS ADR(gShuttles[i]);
							cm ACCESS ADR (gShuttles[i].cm);
							pShuttle.cm.setup.parent.name := 'main';
							pShuttle.cm.setup.nameIdx := i;
							pShuttle.par.shuttleID := i;

							//Chosen action pr shuttle
							CASE i OF
								0:MovementRy;
								3:MovementZ;
								2:MovementRx;
							END_CASE
						END_FOR

				13000..13999:
					em.description := 'Box Program';
					boxProgramTask;

				14000..14999:
					em.description := 'Rotation program';
					rotationTask;
					FOR i := 0 TO NR_OF_WORKSTATIONS DO
						pWorkStations ACCESS ADR (gWorkStations[i]);
						cm ACCESS ADR (gWorkStations[i].cm);
						pWorkStations.cm.setup.parent.name := 'main';
						rotationStation;
					END_FOR

				15000..15999:
					em.description := 'Steelsheet program';
					steelSheetTask;
					FOR i := 0 TO NR_OF_WORKSTATIONS DO
						pWorkStations ACCESS ADR (gWorkStations[i]);
						cm ACCESS ADR (gWorkStations[i].cm);
						pWorkStations.cm.setup.parent.name := 'main';
						steelSheetStation;
					END_FOR

				16000..16999:
					em.description := 'TeachShuttle Program';
					teachShuttleProgram;

				17000..17999:
					em.description := 'Format Change';
					trakModeTask;

				END_CASE

		STATE_STOPPING,STATE_ABORTING:
			ResetInput;
			em.description := 'Power off 6D System';
			CASE em.substate OF
				0:
					IF MC_BR_AsmReadStatus_Acp6D_0.AssemblyReady OR MC_BR_AsmReadStatus_Acp6D_0.AssemblyHoming THEN
						em.substate := 10;
					ELSE
						em.substate := 100;
					END_IF

				10:
					em.description := 'Break all shuttles and shut down the system';
					MC_BR_AsmPowerOff_Acp6D_0.Execute := TRUE;
					IF MC_BR_AsmPowerOff_Acp6D_0.Done THEN
						ResetInput; //Reset all FB
						createShGroup := 0;
						MC_BR_AsmPowerOff_Acp6D_0.Execute := FALSE;
						em.substate := 100;
					END_IF

				100:
					em.description := 'Check if system is off';
					createShGroup := 0;
					em.cmd.sc := TRUE;
			END_CASE

		STATE_CLEARING:
			CASE em.substate OF
				0:
					IF MC_BR_AsmReadStatus_Acp6D_0.AssemblyErrorStop THEN
  						em.substate := 10;
					ELSE
						em.substate := 20;
					END_IF

				10:
					MC_BR_AsmReset_Acp6D_0.Execute := TRUE;
					IF MC_BR_AsmReset_Acp6D_0.Done OR MC_BR_AsmReset_Acp6D_0.Error THEN
  						MC_BR_AsmReset_Acp6D_0.Execute := FALSE;
						em.substate := 20;
					END_IF

				20:
					em.cmd.sc := TRUE;

			END_CASE

		STATE_COMPLETING:
			ResetInput;
			em.description := 'Break all shuttles and clear Motion Buffer';
			CASE em.substate OF
				0:
					em.description := 'Break all shuttles';
					MC_BR_AsmStop_Acp6D_0.Execute := TRUE;
					IF MC_BR_AsmStop_Acp6D_0.Done THEN
						MC_BR_AsmStop_Acp6D_0.Execute := FALSE;
						tempCounter := 0;
						em.substate := 5;
					END_IF

				5:
					FOR i := 0 TO NUM_SHUTTLES DO
						IF gAcp6DCtrl.Status.ShuttleInfo[i].State = mcACP6D_SH_STATE_IDLING OR gAcp6DCtrl.Status.ShuttleInfo[i].State = mcACP6D_SH_STATE_LANDED THEN
						ELSE
							EXIT;
						END_IF
					END_FOR
					IF i > NUM_SHUTTLES THEN
						em.substate := 10;
					END_IF

				10:
					em.description := 'Levitate if any shuttle is landed';
					MC_BR_AsmLevitation_Acp6D_0.Parameters.Speed := 5; //1-5
					MC_BR_AsmLevitation_Acp6D_0.Parameters.Level := 1;
					MC_BR_AsmLevitation_Acp6D_0.Execute := TRUE;
					IF MC_BR_AsmLevitation_Acp6D_0.Done THEN
						MC_BR_AsmLevitation_Acp6D_0.Execute := FALSE;
						em.substate := 100;
					END_IF

				100:
					FOR i := 0 TO NUM_SHUTTLES DO
						IF gAcp6DCtrl.Status.ShuttleInfo[i].State = mcACP6D_SH_STATE_IDLING THEN
						ELSE
							EXIT;
						END_IF
					END_FOR
					IF i > NUM_SHUTTLES THEN
						em.substate := 110;
					END_IF

				110:
					ResetInput;
					em.cmd.reset := TRUE;
					em.cmd.sc := TRUE;
			END_CASE

		ELSE
			em.cmd.sc := TRUE;
	END_CASE

	//Shuttle pos update
	FOR i := 0 TO NUM_SHUTTLES DO
		// check there is a shuttle
		IF gAcp6DCtrl.Status.ShuttleInfo[i].shuttleRef.controlif > 0 THEN
			MC_BR_ShReadInfo_Acp6D_0[i].Shuttle := ADR(gAcp6DCtrl.Status.ShuttleInfo[i].shuttleRef);
			MC_BR_ShReadInfo_Acp6D_0[i].Enable := TRUE;
			gAcp6DCtrl.Status.ShuttleInfo[i].Position := MC_BR_ShReadInfo_Acp6D_0[i].ShuttleInfo.Position;
			gAcp6DCtrl.Status.ShuttleInfo[i].State := MC_BR_ShReadInfo_Acp6D_0[i].ShuttleInfo.State;
			MC_BR_ShReadInfo_Acp6D_0[i]();

			//Turn off system if shuttle is not detected (removed by hand)

			IF em.state = STATE_EXECUTE AND gAcp6DCtrl.Par.modeSelector <> teachProgramEnum AND gAcp6DCtrl.Par.modeSelectorOld <> teachProgramEnum AND NOT shuttleDeativatedLock AND (MC_BR_ShReadInfo_Acp6D_0[i].ShuttleInfo.State = mcACP6D_SH_STATE_RESERVED OR MC_BR_ShReadInfo_Acp6D_0[i].ShuttleInfo.State = mcACP6D_SH_STATE_DISABLED) THEN
				em.cmd.abort := TRUE;
			END_IF
		END_IF
	END_FOR

	em();
	MC_BR_AsmGetShuttle_Acp6D_0();
	MC_BR_AsmReadStatus_Acp6D_0();
	MC_BR_AsmPowerOn_Acp6D_0();
	MC_BR_AsmPowerOff_Acp6D_0();
	MC_BR_AsmStop_Acp6D_0();
	MC_BR_AsmLevitation_Acp6D_0();
	MC_BR_SegPowerOff_Acp6D_0();
	MC_BR_SegPowerOn_Acp6D_0();
	MC_BR_SegBarrierCommand_Acp6D_0();
	MC_BR_AsmGetSegment_Acp6D_0();
	MC_BR_MoveInPlaneAsync_Acp6D_0();
	MC_BR_ShLevitation_Acp6D_0();
	MC_BR_MoveInPlane_Acp6D_0();
	MC_BR_MoveArc_Acp6D_0();
	MC_BR_ShGroupCreate_Acp6D_0();
	MC_BR_ShGroupCreate_Acp6D_1();
	MC_BR_ShGroupCreate_Acp6D_2();
	MC_BR_ShGroupCreate_Acp6D_3();
	MC_BR_ShGroupAddShuttle_Acp6D_0();
	MC_BR_ShGroupCoupleCtrl_Acp6D_0();
	MC_BR_ShGroupGetInfo_Acp6D_0();
	MC_BR_ReadCyclicPosition_Acp6D_0();
	MC_BR_ReadCyclicPosition_Acp6D_1();
	MC_BR_ReadCyclicPosition_Acp6D_2();
	MC_BR_ReadCyclicPosition_Acp6D_3();
	MC_BR_MacroCreate_Acp6D_0();
	MC_BR_Move6D_Acp6D_0();
	MC_BR_MacroRun_Acp6D_0();
	MC_BR_MacroSave_Acp6D_0();
	MC_BR_AsmGetInfo_Acp6D_0();
	MC_BR_RotaryMotionSpin_Acp6D_0();
	MC_BR_ShStop_Acp6D_0();
	MC_BR_RotaryMotion_Acp6D_0();
	TON_watchdog();
	MC_BR_AsmReset_Acp6D_0();

END_PROGRAM

PROGRAM _EXIT
	(* Insert code here *)

END_PROGRAM
```

#### Config.st
```iecst
ACTION config:
	gAcp6DCtrl.Status.Ready := FALSE;
	gameBrain.showHMIButton := FALSE;
	enableButtons := TRUE;

	shuttleStartupInfo[0].initXPos := 0.060;
	shuttleStartupInfo[0].initYPos := 0.060;
	shuttleStartupInfo[1].initXPos := 0.180;
	shuttleStartupInfo[1].initYPos := 0.180;
	shuttleStartupInfo[2].initXPos := 0.300;
	shuttleStartupInfo[2].initYPos := 0.060;
	shuttleStartupInfo[3].initXPos := 0.420;
	shuttleStartupInfo[3].initYPos := 0.180;

END_ACTION
```

#### ResetInput.st
```iecst
ACTION ResetInput:
	MC_BR_AsmPowerOff_Acp6D_0.Execute		:= FALSE;
	MC_BR_AsmPowerOn_Acp6D_0.Execute		:= FALSE;
	MC_BR_ReadCyclicPosition_Acp6D_0.Enable	:= FALSE;
	MC_BR_ReadCyclicPosition_Acp6D_1.Enable	:= FALSE;
	MC_BR_ReadCyclicPosition_Acp6D_2.Enable	:= FALSE;
	MC_BR_ReadCyclicPosition_Acp6D_3.Enable	:= FALSE;
	gAcp6DCtrl.Cmd.PowerOn					:= FALSE;
	gAcp6DCtrl.Cmd.PowerOff					:= FALSE;
	gAcp6DCtrl.Cmd.StartProcess				:= FALSE;
	gAcp6DCtrl.Cmd.StopProcess				:= FALSE;

	ABBRobot.returnBigWeightMovement 		:= FALSE;
	ABBRobot.returnSmallWeightMovement		:= FALSE;
	ABBRobot.startBigWeightMovement			:= FALSE;
	ABBRobot.startSmallWeightMovement		:= FALSE;

	MC_BR_MoveInPlane_Acp6D_0.Execute := FALSE;
	MC_BR_MoveInPlane_Acp6D_0.Parameters.Mode := 0;
	MC_BR_MoveInPlane_Acp6D_0.Parameters.Path := 0;

	FOR i := 0 TO NR_OF_WORKSTATIONS DO
		gWorkStations[i].cm.state := 0;
		gWorkStations[i].MC_BR_ShLevitation_Acp6D_0.Execute := FALSE;
		gWorkStations[i].MC_BR_MoveArc_Acp6D_0.Execute := FALSE;
		gWorkStations[i].MC_BR_MoveInPlane_Acp6D_0.Execute := FALSE;
		gWorkStations[i].MC_BR_RotaryMotion_Acp6D_0.Execute := FALSE;
		gWorkStations[i].MC_BR_RotaryMotionSpin_Acp6D_0.Execute := FALSE;
		gWorkStations[i].MC_BR_Move6D_Acp6D_0.Execute := FALSE;
		gWorkStations[i].MC_BR_MoveShortAxis_Acp6D_0.Execute := FALSE;
		gWorkStations[i].par.ArcMovement := FALSE;
		gWorkStations[i].par.landBeforeProcess := FALSE;
		gWorkStations[i].par.pathRouting := FALSE;
		gWorkStations[i].par.processTime := FALSE;
		gWorkStations[i].par.tempShuttleID := FALSE;
		gWorkStations[i].par.xLocation := FALSE;
		gWorkStations[i].par.yLocation := FALSE;
		gWorkStations[i].par.internalCounter := 0;
		gWorkStations[i].par.tempCounter := 0;
		gWorkStations[i].TON_0.IN := FALSE;
	END_FOR

	FOR i := 0 TO NUM_SHUTTLES DO
		gShuttles[i].function.MC_BR_Move6D_Acp6D_0.Execute := FALSE;
		gShuttles[i].function.MC_BR_MoveInPlane_Acp6D_0.Execute := FALSE;
		gShuttles[i].function.MC_BR_MoveShortAxis_Acp6D_0.Execute := FALSE;
		gShuttles[i].function.TON_0.IN := FALSE;
		gShuttles[i].cm.state := 0;

		//MC_BR_ShReadInfo_Acp6D_0[i].Enable := FALSE;

		//MC_BR_MoveArc_Acp6D_0[i].Execute := FALSE;

		MC_BR_MoveShortAxis_Acp6D_0[i].Execute := FALSE;
	END_FOR

	FOR k := 0 TO 1 DO
		FOR j := 0 TO NUM_SHUTTLES DO
			//MC_BR_ReadCyclicChAxis_Acp6D_0[k,j].Enable := FALSE;
		END_FOR
	END_FOR

	TON_0.IN								:= FALSE;
	MC_BR_MoveArc_Acp6D_0.Execute 			:= FALSE;
	MC_BR_MoveInPlaneAsync_Acp6D_0.Execute	:= FALSE;
	MC_BR_MoveInPlane_Acp6D_0.Execute		:= FALSE;
	//MC_BR_ShReadInfo_Acp6D_0.Execute		:= FALSE;
	MC_BR_ShGroupCreate_Acp6D_0.Execute		:= FALSE;
	MC_BR_ShGroupAddShuttle_Acp6D_0.Execute := FALSE;
	MC_BR_ShGroupCoupleCtrl_Acp6D_0.Execute	:= FALSE;
	MC_BR_ShGroupGetInfo_Acp6D_0.Execute	:= FALSE;
	MC_BR_SegPowerOff_Acp6D_0.Execute		:= FALSE;
	MC_BR_SegPowerOn_Acp6D_0.Execute		:= FALSE;
	MC_BR_SegBarrierCommand_Acp6D_0.Execute	:= FALSE;
	MC_BR_RotaryMotion_Acp6D_0.Execute 		:= FALSE;
	MC_BR_ShStop_Acp6D_0.Execute			:= FALSE;
	MC_BR_RotaryMotionSpin_Acp6D_0.Execute	:= FALSE;
	//MC_BR_MacroList_Acp6D_0.Execute			:= FALSE;
	//MC_BR_MacroLoad_Acp6D_0.Execute			:= FALSE;
	//MC_BR_MoveShortAxis_Acp6D_0.Execute		:= FALSE;
	//MC_BR_PlanetCtrl_Acp6D_0.Execute		:= FALSE;
	MC_BR_Move6D_Acp6D_0.Execute 			:= FALSE;
	MC_BR_ShLevitation_Acp6D_0.Execute		:= FALSE;
	MC_BR_AsmLevitation_Acp6D_0.Execute 	:= FALSE;
	MC_BR_AsmGetShuttle_Acp6D_0.Enable 		:= FALSE;
	MC_BR_AsmGetSegment_Acp6D_0.Enable 		:= FALSE;

	//MC_BR_MacroList_Acp6D_0();
	//MC_BR_MacroLoad_Acp6D_0();

END_ACTION
```

#### shuttleGroups.st
```iecst
ACTION shuttleGroups:
	CASE createShGroup OF
		0:
			//Create First shuttle Group
			MC_BR_ShGroupCreate_Acp6D_0.Execute := TRUE;
			IF MC_BR_ShGroupCreate_Acp6D_0.Done THEN
				shGroupShuttle1_2 := ADR(MC_BR_ShGroupCreate_Acp6D_0.ShuttleGroup);
				MC_BR_ShGroupCreate_Acp6D_0.Execute := FALSE;
				createShGroup := 10;
			END_IF

		10:
			//Add shuttles to new group
			MC_BR_ShGroupAddShuttle_Acp6D_0.ShuttleGroup := shGroupShuttle1_2;
			MC_BR_ShGroupAddShuttle_Acp6D_0.Parameters.ShuttleList[0].Shuttle := ADR(gAcp6DCtrl.Status.ShuttleInfo[0].shuttleRef);
			MC_BR_ShGroupAddShuttle_Acp6D_0.Parameters.ShuttleList[1].Shuttle := ADR(gAcp6DCtrl.Status.ShuttleInfo[1].shuttleRef);
			MC_BR_ShGroupAddShuttle_Acp6D_0.Execute := TRUE;
			IF MC_BR_ShGroupAddShuttle_Acp6D_0.Done THEN
				MC_BR_ShGroupAddShuttle_Acp6D_0.Execute := FALSE;
				createShGroup := 15;
			END_IF

		15:
			//dummy scan
			IF NOT MC_BR_ShGroupAddShuttle_Acp6D_0.Done THEN
				createShGroup := 20;
			END_IF

		20:
			//Create Second shuttle Group
			MC_BR_ShGroupCreate_Acp6D_1.Execute := TRUE;
			IF MC_BR_ShGroupCreate_Acp6D_1.Done THEN
				shGroupShuttle3_4 := ADR(MC_BR_ShGroupCreate_Acp6D_1.ShuttleGroup);
				MC_BR_ShGroupCreate_Acp6D_1.Execute := FALSE;
				createShGroup := 30;
			END_IF

		30:
			//Add shuttles to new group
			MC_BR_ShGroupAddShuttle_Acp6D_0.ShuttleGroup := shGroupShuttle3_4;
			MC_BR_ShGroupAddShuttle_Acp6D_0.Parameters.ShuttleList[0].Shuttle := ADR(gAcp6DCtrl.Status.ShuttleInfo[2].shuttleRef);
			MC_BR_ShGroupAddShuttle_Acp6D_0.Parameters.ShuttleList[1].Shuttle := ADR(gAcp6DCtrl.Status.ShuttleInfo[3].shuttleRef);
			MC_BR_ShGroupAddShuttle_Acp6D_0.Execute := TRUE;
			IF MC_BR_ShGroupAddShuttle_Acp6D_0.Done THEN
				MC_BR_ShGroupAddShuttle_Acp6D_0.Execute := FALSE;
				createShGroup := 40;
			END_IF

		40:
			//Create third shuttle Group
			MC_BR_ShGroupCreate_Acp6D_2.Execute := TRUE;
			IF MC_BR_ShGroupCreate_Acp6D_2.Done THEN
				shGroupShuttle1_4 := ADR(MC_BR_ShGroupCreate_Acp6D_2.ShuttleGroup);
				MC_BR_ShGroupCreate_Acp6D_2.Execute := FALSE;
				createShGroup := 50;
			END_IF

		50:
			//Add shuttles to new group
			MC_BR_ShGroupAddShuttle_Acp6D_0.ShuttleGroup := shGroupShuttle1_4;
			MC_BR_ShGroupAddShuttle_Acp6D_0.Parameters.ShuttleList[0].Shuttle := ADR(gAcp6DCtrl.Status.ShuttleInfo[0].shuttleRef);
			MC_BR_ShGroupAddShuttle_Acp6D_0.Parameters.ShuttleList[1].Shuttle := ADR(gAcp6DCtrl.Status.ShuttleInfo[3].shuttleRef);
			MC_BR_ShGroupAddShuttle_Acp6D_0.Execute := TRUE;
			IF MC_BR_ShGroupAddShuttle_Acp6D_0.Done THEN
				MC_BR_ShGroupAddShuttle_Acp6D_0.Execute := FALSE;
				createShGroup := 60;
			END_IF

		60:
			//Create fourth shuttle Group
			MC_BR_ShGroupCreate_Acp6D_3.Execute := TRUE;
			IF MC_BR_ShGroupCreate_Acp6D_3.Done THEN
				shGroupShuttle2_3 := ADR(MC_BR_ShGroupCreate_Acp6D_3.ShuttleGroup);
				MC_BR_ShGroupCreate_Acp6D_3.Execute := FALSE;
				createShGroup := 70;
			END_IF

		70:
			//Add shuttles to new group
			MC_BR_ShGroupAddShuttle_Acp6D_0.ShuttleGroup := shGroupShuttle2_3;
			MC_BR_ShGroupAddShuttle_Acp6D_0.Parameters.ShuttleList[0].Shuttle := ADR(gAcp6DCtrl.Status.ShuttleInfo[1].shuttleRef);
			MC_BR_ShGroupAddShuttle_Acp6D_0.Parameters.ShuttleList[1].Shuttle := ADR(gAcp6DCtrl.Status.ShuttleInfo[2].shuttleRef);
			MC_BR_ShGroupAddShuttle_Acp6D_0.Execute := TRUE;
			IF MC_BR_ShGroupAddShuttle_Acp6D_0.Done THEN
				MC_BR_ShGroupAddShuttle_Acp6D_0.Execute := FALSE;
				createShGroup := 80;
			END_IF
	END_CASE
END_ACTION
ACTION macroCreatorAction:
	CASE macroCreater OF
		0:
			MC_BR_MacroCreate_Acp6D_0.Parameters.Name := 'shuttleWave';
			MC_BR_MacroCreate_Acp6D_0.Execute := TRUE;
			IF MC_BR_MacroCreate_Acp6D_0.Done THEN
				MC_BR_MacroCreate_Acp6D_0.Execute := FALSE;
				macroCreater := 10;
			END_IF

		10:
			MC_BR_MoveInPlane_Acp6D_0.Shuttle := ADR(MC_BR_MacroCreate_Acp6D_0.MacroShuttle);
			MC_BR_MoveInPlane_Acp6D_0.Parameters.Position.X := 0.0;
			MC_BR_MoveInPlane_Acp6D_0.Parameters.Position.Y := 0.060;
			MC_BR_MoveInPlane_Acp6D_0.Parameters.Velocity := gAcp6DCtrl.Par.Velocity;
			MC_BR_MoveInPlane_Acp6D_0.Parameters.Acceleration := gAcp6DCtrl.Par.Acceleration;
			MC_BR_MoveInPlane_Acp6D_0.Parameters.Mode := 1; //Relative
			MC_BR_MoveInPlane_Acp6D_0.Parameters.Path := 0; //Y then X
			MC_BR_MoveInPlane_Acp6D_0.Execute := TRUE;
			IF MC_BR_MoveInPlane_Acp6D_0.Acknowledge THEN
				MC_BR_MoveInPlane_Acp6D_0.Execute := FALSE;
				macroCreater := 20;
			END_IF

		20:
			MC_BR_MoveInPlane_Acp6D_0.Shuttle := ADR(MC_BR_MacroCreate_Acp6D_0.MacroShuttle);
			MC_BR_MoveInPlane_Acp6D_0.Parameters.Position.X := 0.0;
			MC_BR_MoveInPlane_Acp6D_0.Parameters.Position.Y := -0.120;
			MC_BR_MoveInPlane_Acp6D_0.Parameters.Velocity := gAcp6DCtrl.Par.Velocity;
			MC_BR_MoveInPlane_Acp6D_0.Parameters.Acceleration := gAcp6DCtrl.Par.Acceleration;
			MC_BR_MoveInPlane_Acp6D_0.Parameters.Mode := 1; //Relative
			MC_BR_MoveInPlane_Acp6D_0.Parameters.Path := 0; //Y then X
			MC_BR_MoveInPlane_Acp6D_0.Execute := TRUE;
			IF MC_BR_MoveInPlane_Acp6D_0.Acknowledge THEN
				MC_BR_MoveInPlane_Acp6D_0.Execute := FALSE;
				macroCreater := 30;
			END_IF

		30:
			MC_BR_MoveInPlane_Acp6D_0.Shuttle := ADR(MC_BR_MacroCreate_Acp6D_0.MacroShuttle);
			MC_BR_MoveInPlane_Acp6D_0.Parameters.Position.X := 0.0;
			MC_BR_MoveInPlane_Acp6D_0.Parameters.Position.Y := 0.120;
			MC_BR_MoveInPlane_Acp6D_0.Parameters.Velocity := gAcp6DCtrl.Par.Velocity;
			MC_BR_MoveInPlane_Acp6D_0.Parameters.Acceleration := gAcp6DCtrl.Par.Acceleration;
			MC_BR_MoveInPlane_Acp6D_0.Parameters.Mode := 1; //Relative
			MC_BR_MoveInPlane_Acp6D_0.Parameters.Path := 0; //Y then X
			MC_BR_MoveInPlane_Acp6D_0.Execute := TRUE;
			IF MC_BR_MoveInPlane_Acp6D_0.Acknowledge THEN
				MC_BR_MoveInPlane_Acp6D_0.Execute := FALSE;
				macroCreater := 40;
			END_IF

		40:
			MC_BR_MoveInPlane_Acp6D_0.Shuttle := ADR(MC_BR_MacroCreate_Acp6D_0.MacroShuttle);
			MC_BR_MoveInPlane_Acp6D_0.Parameters.Position.X := 0.0;
			MC_BR_MoveInPlane_Acp6D_0.Parameters.Position.Y := -0.120;
			MC_BR_MoveInPlane_Acp6D_0.Parameters.Velocity := gAcp6DCtrl.Par.Velocity;
			MC_BR_MoveInPlane_Acp6D_0.Parameters.Acceleration := gAcp6DCtrl.Par.Acceleration;
			MC_BR_MoveInPlane_Acp6D_0.Parameters.Mode := 1; //Relative
			MC_BR_MoveInPlane_Acp6D_0.Parameters.Path := 0; //Y then X
			MC_BR_MoveInPlane_Acp6D_0.Execute := TRUE;
			IF MC_BR_MoveInPlane_Acp6D_0.Acknowledge THEN
				MC_BR_MoveInPlane_Acp6D_0.Execute := FALSE;
				macroCreater := 50;
			END_IF

		50:
			MC_BR_MoveInPlane_Acp6D_0.Shuttle := ADR(MC_BR_MacroCreate_Acp6D_0.MacroShuttle);
			MC_BR_MoveInPlane_Acp6D_0.Parameters.Position.X := 0.0;
			MC_BR_MoveInPlane_Acp6D_0.Parameters.Position.Y := 0.120;
			MC_BR_MoveInPlane_Acp6D_0.Parameters.Velocity := gAcp6DCtrl.Par.Velocity;
			MC_BR_MoveInPlane_Acp6D_0.Parameters.Acceleration := gAcp6DCtrl.Par.Acceleration;
			MC_BR_MoveInPlane_Acp6D_0.Parameters.Mode := 1; //Relative
			MC_BR_MoveInPlane_Acp6D_0.Parameters.Path := 0; //Y then X
			MC_BR_MoveInPlane_Acp6D_0.Execute := TRUE;
			IF MC_BR_MoveInPlane_Acp6D_0.Acknowledge THEN
				MC_BR_MoveInPlane_Acp6D_0.Execute := FALSE;
				macroCreater := 60;
			END_IF

		60:
			MC_BR_MacroSave_Acp6D_0.Shuttle := ADR(MC_BR_MacroCreate_Acp6D_0.MacroShuttle);
			MC_BR_MacroSave_Acp6D_0.Execute := TRUE;
			IF MC_BR_MacroSave_Acp6D_0.Done THEN
				MC_BR_MacroSave_Acp6D_0.Execute := FALSE;
				macroCreater := 70;
			END_IF

		70:
			//nothing
	END_CASE

END_ACTION
```
